KUKA KRL program: EPS_2_26115_SA7000_A_20260219035533.src

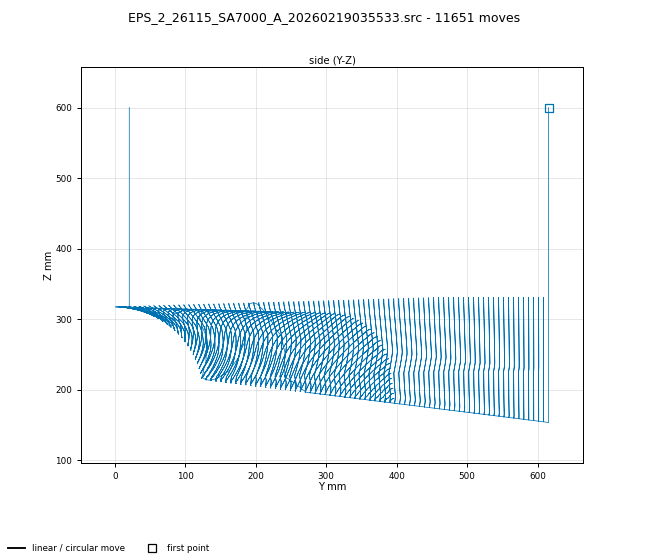
[picture p0: tool path of EPS_2_26115_SA7000_A_20260219035533.src, 11651 of 11653 moves have a stored position in this frame; points joined in program order, loops and branches not executed]
&ACCESS RVP
&REL 4
&COMMENT QRS 19112012
&PARAM EDITMASK = *
DEF PART()
EXT BAS (BAS_COMMAND :IN,REAL :IN )
INT I
BAS (#INITMOV,0 )

;KUKA QRS Post kuka4.cps  Date:22-06-2017 !

File_ID=3055

QRS_PRE_INIT()

;Init var - Until changes are made in qrs_pre_init
Outlet_Square_prg=0
Inlet_1_Square_prg=0
Inlet_2_Square_prg=0
Inlet_3_Square_prg=0
Inlet_4_Square_prg=0
Inlet_5_Square_prg=0

Outlet_1={X 0.000, Y 460.000, Z 230.500, B 0.000, E1 0.000 }
Inlet_1={X 0.000, Y 565.490, Z 205.500, B 0.000, E1 180.000 }
Outlet_1_type=201
Inlet_1_type=0
;QRS#1=Sidecore dimensions
;QRS#2=200-8" PVC SDR 35 Cut Back
;QRS#3=DeadEnd 201
;QRS#4=
;QRS#5=
;QRS#6=
;QRS#7=
;QRS#8=
;QRS#9=12-08 PSX
;QRS#10=

;QRS#11=
;QRS#12=
;QRS#13=
;QRS#14=
;QRS#15=
;QRS#16=1220x127x610 2'
;QRS#17=EPS Height
;QRS#18=331
;QRS#19=*
;QRS#20= UPDATED VERSION 22-06-2017
;QRS#21=*
Outlet_Square=0100
Inlet_1_Square=00
Inlet_2_Square=0
Inlet_3_Square=0
Inlet_4_Square=0
Inlet_5_Square=0
Mill_Square=1
Outlet_Square_Prg=214
Inlet_1_Square_prg=0

QRS_INIT()

$ADVANCE=5

; T1
PTP {E1 173.609,E2 173.609}
PTP {X 0,Y 615.488,A -85,B 0,C 180,E1 173.609,E2 173.609,E3 0,E4 0,E5 0,E6 0}
QRS_SPEED_INIT()
LIN {X 0,Y 615.488,Z 600,A -85,B 0,C 180,E1 173.609,E2 173.609,E3 0,E4 0,E5 0,E6 0} C_VEL
LIN {X 0,Y 615.488,Z 163.366,A -85,B 0,C 180,E1 173.609,E2 173.609} C_VEL
LIN {X 0,Y 615.488,Z 155.185,A -85,B 0,C 180,E1 173.609,E2 173.609} C_VEL
LIN {X 0,Y 615.477,Z 153.185,A -85,B 0,C 180,E1 173.423,E2 173.423} C_VEL
LIN {X 0,Y 615.491,Z 153.195,A -85,B 0,C 180,E1 170.802,E2 170.802} C_VEL
LIN {X 0,Y 615.463,Z 153.193,A -85,B 0,C 180,E1 168.139,E2 168.139} C_VEL
LIN {X 0,Y 615.491,Z 153.184,A -85,B 0,C 180,E1 165.451,E2 165.451} C_VEL
LIN {X 0,Y 615.488,Z 153.199,A -85,B 0,C 180,E1 162.73,E2 162.73} C_VEL
LIN {X 0,Y 615.475,Z 153.186,A -85,B 0,C 180,E1 159.967,E2 159.967} C_VEL
LIN {X 0,Y 615.485,Z 153.198,A -85,B 0,C 180,E1 157.156,E2 157.156} C_VEL
LIN {X 0,Y 615.467,Z 153.19,A -85,B 0,C 180,E1 154.433,E2 154.433} C_VEL
LIN {X 0,Y 615.482,Z 153.184,A -85,B 0,C 180,E1 152.085,E2 152.085} C_VEL
LIN {X 0,Y 615.486,Z 153.198,A -85,B 0,C 180,E1 149.081,E2 149.081} C_VEL
LIN {X 0,Y 615.474,Z 153.186,A -85,B 0,C 180,E1 146.466,E2 146.466} C_VEL
LIN {X 0,Y 615.488,Z 153.184,A -85,B 0,C 180,E1 144.165,E2 144.165} C_VEL
LIN {X 0,Y 615.484,Z 153.189,A -85,B 0,C 180,E1 141.932,E2 141.932} C_VEL
LIN {X 0,Y 615.488,Z 153.198,A -85,B 0,C 180,E1 139.394,E2 139.394} C_VEL
LIN {X 0,Y 615.477,Z 153.186,A -85,B 0,C 180,E1 136.755,E2 136.755} C_VEL
LIN {X 0,Y 615.481,Z 153.194,A -85,B 0,C 180,E1 133.997,E2 133.997} C_VEL
LIN {X 0,Y 615.478,Z 153.195,A -85,B 0,C 180,E1 131.474,E2 131.474} C_VEL
LIN {X 0,Y 615.478,Z 153.185,A -85,B 0,C 180,E1 128.904,E2 128.904} C_VEL
LIN {X 0,Y 615.483,Z 153.189,A -85,B 0,C 180,E1 126.424,E2 126.424} C_VEL
LIN {X 0,Y 615.491,Z 153.201,A -85,B 0,C 180,E1 124.021,E2 124.021} C_VEL
LIN {X 0,Y 615.481,Z 153.184,A -85,B 0,C 180,E1 121.086,E2 121.086} C_VEL
LIN {X 0,Y 615.484,Z 153.194,A -85,B 0,C 180,E1 118.451,E2 118.451} C_VEL
LIN {X 0,Y 615.472,Z 153.191,A -85,B 0,C 180,E1 115.716,E2 115.716} C_VEL
LIN {X 0,Y 615.478,Z 153.186,A -85,B 0,C 180,E1 113.556,E2 113.556} C_VEL
LIN {X 0,Y 615.482,Z 153.193,A -85,B 0,C 180,E1 110.731,E2 110.731} C_VEL
LIN {X 0,Y 615.475,Z 153.191,A -85,B 0,C 180,E1 107.957,E2 107.957} C_VEL
LIN {X 0,Y 615.484,Z 153.186,A -85,B 0,C 180,E1 105.226,E2 105.226} C_VEL
LIN {X 0,Y 615.491,Z 153.199,A -85,B 0,C 180,E1 102.53,E2 102.53} C_VEL
LIN {X 0,Y 615.486,Z 153.184,A -85,B 0,C 180,E1 99.862,E2 99.862} C_VEL
LIN {X 0,Y 615.479,Z 153.191,A -85,B 0,C 180,E1 97.216,E2 97.216} C_VEL
LIN {X 0,Y 615.482,Z 153.195,A -85,B 0,C 180,E1 94.585,E2 94.585} C_VEL
LIN {X 0,Y 615.498,Z 153.181,A -85,B 0,C 180,E1 91.963,E2 91.963} C_VEL
LIN {X 0,Y 615.481,Z 153.194,A -85,B 0,C 180,E1 89.346,E2 89.346} C_VEL
LIN {X 0,Y 615.48,Z 153.193,A -85,B 0,C 180,E1 86.727,E2 86.727} C_VEL
LIN {X 0,Y 615.492,Z 153.182,A -85,B 0,C 180,E1 84.102,E2 84.102} C_VEL
LIN {X 0,Y 615.485,Z 153.196,A -85,B 0,C 180,E1 81.463,E2 81.463} C_VEL
LIN {X 0,Y 615.48,Z 153.189,A -85,B 0,C 180,E1 78.807,E2 78.807} C_VEL
LIN {X 0,Y 615.476,Z 153.188,A -85,B 0,C 180,E1 76.07,E2 76.07} C_VEL
LIN {X 0,Y 615.487,Z 153.2,A -85,B 0,C 180,E1 73.414,E2 73.414} C_VEL
LIN {X 0,Y 615.486,Z 153.183,A -85,B 0,C 180,E1 70.662,E2 70.662} C_VEL
LIN {X 0,Y 615.483,Z 153.197,A -85,B 0,C 180,E1 67.864,E2 67.864} C_VEL
LIN {X 0,Y 615.489,Z 153.184,A -85,B 0,C 180,E1 65.009,E2 65.009} C_VEL
LIN {X 0,Y 615.488,Z 153.183,A -85,B 0,C 180,E1 62.823,E2 62.823} C_VEL
LIN {X 0,Y 615.478,Z 153.194,A -85,B 0,C 180,E1 60.206,E2 60.206} C_VEL
LIN {X 0,Y 615.482,Z 153.191,A -85,B 0,C 180,E1 57.543,E2 57.543} C_VEL
LIN {X 0,Y 615.496,Z 153.181,A -85,B 0,C 180,E1 55.186,E2 55.186} C_VEL
LIN {X 0,Y 615.473,Z 153.189,A -85,B 0,C 180,E1 52.757,E2 52.757} C_VEL
LIN {X 0,Y 615.486,Z 153.194,A -85,B 0,C 180,E1 49.911,E2 49.911} C_VEL
LIN {X 0,Y 615.487,Z 153.186,A -85,B 0,C 180,E1 47.648,E2 47.648} C_VEL
LIN {X 0,Y 615.471,Z 153.19,A -85,B 0,C 180,E1 44.931,E2 44.931} C_VEL
LIN {X 0,Y 615.485,Z 153.192,A -85,B 0,C 180,E1 42.081,E2 42.081} C_VEL
LIN {X 0,Y 615.495,Z 153.182,A -85,B 0,C 180,E1 39.749,E2 39.749} C_VEL
LIN {X 0,Y 615.474,Z 153.194,A -85,B 0,C 180,E1 36.936,E2 36.936} C_VEL
LIN {X 0,Y 615.49,Z 153.2,A -85,B 0,C 180,E1 34.702,E2 34.702} C_VEL
LIN {X 0,Y 615.479,Z 153.185,A -85,B 0,C 180,E1 31.685,E2 31.685} C_VEL
LIN {X 0,Y 615.468,Z 153.191,A -85,B 0,C 180,E1 29.407,E2 29.407} C_VEL
LIN {X 0,Y 615.484,Z 153.198,A -85,B 0,C 180,E1 27.046,E2 27.046} C_VEL
LIN {X 0,Y 615.483,Z 153.184,A -85,B 0,C 180,E1 24.009,E2 24.009} C_VEL
LIN {X 0,Y 615.471,Z 153.194,A -85,B 0,C 180,E1 21.432,E2 21.432} C_VEL
LIN {X 0,Y 615.49,Z 153.187,A -85,B 0,C 180,E1 18.608,E2 18.608} C_VEL
LIN {X 0,Y 615.466,Z 153.19,A -85,B 0,C 180,E1 15.905,E2 15.905} C_VEL
LIN {X 0,Y 615.495,Z 153.198,A -85,B 0,C 180,E1 13.201,E2 13.201} C_VEL
LIN {X 0,Y 615.483,Z 153.184,A -85,B 0,C 180,E1 10.527,E2 10.527} C_VEL
LIN {X 0,Y 615.466,Z 153.194,A -85,B 0,C 180,E1 7.876,E2 7.876} C_VEL
LIN {X 0,Y 615.49,Z 153.193,A -85,B 0,C 180,E1 5.241,E2 5.241} C_VEL
LIN {X 0,Y 615.474,Z 153.186,A -85,B 0,C 180,E1 2.618,E2 2.618} C_VEL
LIN {X 0,Y 615.473,Z 153.196,A -85,B 0,C 180,E1 0,E2 0} C_VEL
LIN {X 0,Y 615.49,Z 153.19,A -85,B 0,C 180,E1 -2.618,E2 -2.618} C_VEL
LIN {X 0,Y 615.467,Z 153.188,A -85,B 0,C 180,E1 -5.242,E2 -5.242} C_VEL
LIN {X 0,Y 615.48,Z 153.197,A -85,B 0,C 180,E1 -7.876,E2 -7.876} C_VEL
LIN {X 0,Y 615.475,Z 153.186,A -85,B 0,C 180,E1 -10.887,E2 -10.887} C_VEL
LIN {X 0,Y 615.46,Z 153.191,A -85,B 0,C 180,E1 -13.202,E2 -13.202} C_VEL
LIN {X 0,Y 615.488,Z 153.2,A -85,B 0,C 180,E1 -15.905,E2 -15.905} C_VEL
LIN {X 0,Y 615.474,Z 153.186,A -85,B 0,C 180,E1 -18.647,E2 -18.647} C_VEL
LIN {X 0,Y 615.476,Z 153.197,A -85,B 0,C 180,E1 -21.433,E2 -21.433} C_VEL
LIN {X 0,Y 615.485,Z 153.186,A -85,B 0,C 180,E1 -24.272,E2 -24.272} C_VEL
LIN {X 0,Y 615.469,Z 153.187,A -85,B 0,C 180,E1 -26.445,E2 -26.445} C_VEL
LIN {X 0,Y 615.455,Z 153.191,A -85,B 0,C 180,E1 -28.66,E2 -28.66} C_VEL
LIN {X 0,Y 615.471,Z 153.197,A -85,B 0,C 180,E1 -31.085,E2 -31.085} C_VEL
LIN {X 0,Y 615.48,Z 153.186,A -85,B 0,C 180,E1 -34.023,E2 -34.023} C_VEL
LIN {X 0,Y 615.455,Z 153.191,A -85,B 0,C 180,E1 -36.427,E2 -36.427} C_VEL
LIN {X 0,Y 615.49,Z 153.199,A -85,B 0,C 180,E1 -39.063,E2 -39.063} C_VEL
LIN {X 0,Y 615.493,Z 153.189,A -85,B 0,C 180,E1 -41.474,E2 -41.474} C_VEL
LIN {X 0,Y 615.454,Z 153.191,A -85,B 0,C 180,E1 -44.153,E2 -44.153} C_VEL
LIN {X 0,Y 615.489,Z 153.201,A -85,B 0,C 180,E1 -46.953,E2 -46.953} C_VEL
LIN {X 0,Y 615.481,Z 153.336,A -85,B 0,C 180,E1 -48.716,E2 -48.716} C_VEL
LIN {X 0,Y 615.489,Z 158.318,A -85,B 0,C 180,E1 -51.096,E2 -51.096} C_VEL
LIN {X 0,Y 615.47,Z 163.694,A -85,B 0,C 180,E1 -53.575,E2 -53.575} C_VEL
LIN {X 0,Y 615.471,Z 169.069,A -85,B 0,C 180,E1 -55.978,E2 -55.978} C_VEL
LIN {X 0,Y 615.484,Z 175.834,A -85,B 0,C 180,E1 -58.915,E2 -58.915} C_VEL
LIN {X 0,Y 615.48,Z 182.098,A -85,B 0,C 180,E1 -61.552,E2 -61.552} C_VEL
LIN {X 0,Y 615.472,Z 188.743,A -85,B 0,C 180,E1 -64.284,E2 -64.284} C_VEL
LIN {X 0,Y 615.474,Z 194.107,A -85,B 0,C 180,E1 -66.444,E2 -66.444} C_VEL
LIN {X 0,Y 615.49,Z 201.253,A -85,B 0,C 180,E1 -69.27,E2 -69.27} C_VEL
LIN {X 0,Y 615.457,Z 208.403,A -85,B 0,C 180,E1 -72.042,E2 -72.042} C_VEL
LIN {X 0,Y 615.495,Z 215.538,A -85,B 0,C 180,E1 -74.774,E2 -74.774} C_VEL
LIN {X 0,Y 615.438,Z 222.684,A -85,B 0,C 180,E1 -77.469,E2 -77.469} C_VEL
LIN {X 0,Y 615.49,Z 225.076,A -85,B 0,C 180,E1 -78.369,E2 -78.369} C_VEL
LIN {X 0,Y 615.481,Z 240.867,A -85,B 0,C 180,E1 -78.724,E2 -78.724} C_VEL
LIN {X 0,Y 615.44,Z 253.271,A -85,B 0,C 180,E1 -79.136,E2 -79.136} C_VEL
LIN {X 0,Y 615.434,Z 264.489,A -85,B 0,C 180,E1 -79.639,E2 -79.639} C_VEL
LIN {X 0,Y 615.485,Z 275.998,A -85,B 0,C 180,E1 -80.304,E2 -80.304} C_VEL
LIN {X 0,Y 615.499,Z 286.343,A -85,B 0,C 180,E1 -81.05,E2 -81.05} C_VEL
LIN {X 0,Y 615.497,Z 294.813,A -85,B 0,C 180,E1 -81.794,E2 -81.794} C_VEL
LIN {X 0,Y 615.498,Z 302.607,A -85,B 0,C 180,E1 -82.62,E2 -82.62} C_VEL
LIN {X 0,Y 615.496,Z 310.204,A -85,B 0,C 180,E1 -83.608,E2 -83.608} C_VEL
LIN {X 0,Y 615.498,Z 317.205,A -85,B 0,C 180,E1 -84.759,E2 -84.759} C_VEL
LIN {X 0,Y 615.493,Z 321.852,A -85,B 0,C 180,E1 -85.744,E2 -85.744} C_VEL
LIN {X 0,Y 615.494,Z 325.399,A -85,B 0,C 180,E1 -86.727,E2 -86.727} C_VEL
LIN {X 0,Y 615.497,Z 327.233,A -85,B 0,C 180,E1 -87.382,E2 -87.382} C_VEL
LIN {X 0,Y 615.5,Z 328.608,A -85,B 0,C 180,E1 -88.037,E2 -88.037} C_VEL
LIN {X 0,Y 615.496,Z 330.173,A -85,B 0,C 180,E1 -89.346,E2 -89.346} C_VEL
LIN {X 0,Y 615.494,Z 330.389,A -85,B 0,C 180,E1 -90,E2 -90} C_VEL
LIN {X 0,Y 615.495,Z 329.58,A -85,B 0,C 180,E1 -91.309,E2 -91.309} C_VEL
LIN {X 0,Y 615.5,Z 328.608,A -85,B 0,C 180,E1 -91.963,E2 -91.963} C_VEL
LIN {X 0,Y 615.497,Z 327.233,A -85,B 0,C 180,E1 -92.618,E2 -92.618} C_VEL
LIN {X 0,Y 615.496,Z 324.35,A -85,B 0,C 180,E1 -93.601,E2 -93.601} C_VEL
LIN {X 0,Y 615.498,Z 320.442,A -85,B 0,C 180,E1 -94.584,E2 -94.584} C_VEL
LIN {X 0,Y 615.499,Z 315.405,A -85,B 0,C 180,E1 -95.57,E2 -95.57} C_VEL
LIN {X 0,Y 615.497,Z 308.87,A -85,B 0,C 180,E1 -96.583,E2 -96.583} C_VEL
LIN {X 0,Y 615.497,Z 301.134,A -85,B 0,C 180,E1 -97.545,E2 -97.545} C_VEL
LIN {X 0,Y 615.498,Z 293.046,A -85,B 0,C 180,E1 -98.371,E2 -98.371} C_VEL
LIN {X 0,Y 615.499,Z 283.169,A -85,B 0,C 180,E1 -99.198,E2 -99.198} C_VEL
LIN {X 0,Y 615.464,Z 271.988,A -85,B 0,C 180,E1 -99.945,E2 -99.945} C_VEL
LIN {X 0,Y 615.43,Z 261.035,A -85,B 0,C 180,E1 -100.528,E2 -100.528} C_VEL
LIN {X 0,Y 615.453,Z 248.835,A -85,B 0,C 180,E1 -101.029,E2 -101.029} C_VEL
LIN {X 0,Y 615.495,Z 236.071,A -85,B 0,C 180,E1 -101.401,E2 -101.401} C_VEL
LIN {X 0,Y 615.49,Z 225.076,A -85,B 0,C 180,E1 -101.631,E2 -101.631} C_VEL
LIN {X 0,Y 615.457,Z 219,A -85,B 0,C 180,E1 -103.92,E2 -103.92} C_VEL
LIN {X 0,Y 615.451,Z 212.413,A -85,B 0,C 180,E1 -106.419,E2 -106.419} C_VEL
LIN {X 0,Y 615.487,Z 204.835,A -85,B 0,C 180,E1 -109.338,E2 -109.338} C_VEL
LIN {X 0,Y 615.47,Z 197.68,A -85,B 0,C 180,E1 -112.137,E2 -112.137} C_VEL
LIN {X 0,Y 615.49,Z 190.536,A -85,B 0,C 180,E1 -114.991,E2 -114.991} C_VEL
LIN {X 0,Y 615.489,Z 185.167,A -85,B 0,C 180,E1 -117.177,E2 -117.177} C_VEL
LIN {X 0,Y 615.49,Z 178.875,A -85,B 0,C 180,E1 -119.794,E2 -119.794} C_VEL
LIN {X 0,Y 615.471,Z 172.648,A -85,B 0,C 180,E1 -122.458,E2 -122.458} C_VEL
LIN {X 0,Y 615.496,Z 167.272,A -85,B 0,C 180,E1 -124.814,E2 -124.814} C_VEL
LIN {X 0,Y 615.489,Z 161.901,A -85,B 0,C 180,E1 -127.241,E2 -127.241} C_VEL
LIN {X 0,Y 615.454,Z 156.533,A -85,B 0,C 180,E1 -129.752,E2 -129.752} C_VEL
LIN {X 0,Y 615.474,Z 153.198,A -85,B 0,C 180,E1 -131.379,E2 -131.379} C_VEL
LIN {X 0,Y 615.461,Z 153.189,A -85,B 0,C 180,E1 -134.151,E2 -134.151} C_VEL
LIN {X 0,Y 615.487,Z 153.202,A -85,B 0,C 180,E1 -136.952,E2 -136.952} C_VEL
LIN {X 0,Y 615.459,Z 153.195,A -85,B 0,C 180,E1 -139.391,E2 -139.391} C_VEL
LIN {X 0,Y 615.472,Z 153.187,A -85,B 0,C 180,E1 -141.989,E2 -141.989} C_VEL
LIN {X 0,Y 615.493,Z 153.19,A -85,B 0,C 180,E1 -144.384,E2 -144.384} C_VEL
LIN {X 0,Y 615.485,Z 153.2,A -85,B 0,C 180,E1 -146.763,E2 -146.763} C_VEL
LIN {X 0,Y 615.461,Z 153.195,A -85,B 0,C 180,E1 -149.078,E2 -149.078} C_VEL
LIN {X 0,Y 615.464,Z 153.188,A -85,B 0,C 180,E1 -151.552,E2 -151.552} C_VEL
LIN {X 0,Y 615.499,Z 153.2,A -85,B 0,C 180,E1 -154.427,E2 -154.427} C_VEL
LIN {X 0,Y 615.458,Z 153.191,A -85,B 0,C 180,E1 -157.154,E2 -157.154} C_VEL
LIN {X 0,Y 615.492,Z 153.191,A -85,B 0,C 180,E1 -159.967,E2 -159.967} C_VEL
LIN {X 0,Y 615.461,Z 153.193,A -85,B 0,C 180,E1 -162.728,E2 -162.728} C_VEL
LIN {X 0,Y 615.489,Z 153.185,A -85,B 0,C 180,E1 -165.451,E2 -165.451} C_VEL
LIN {X 0,Y 615.483,Z 153.2,A -85,B 0,C 180,E1 -168.139,E2 -168.139} C_VEL
LIN {X 0,Y 615.463,Z 153.189,A -85,B 0,C 180,E1 -170.801,E2 -170.801} C_VEL
LIN {X 0,Y 615.489,Z 153.189,A -85,B 0,C 180,E1 -173.443,E2 -173.443} C_VEL
LIN {X 0,Y 615.475,Z 153.196,A -85,B 0,C 180,E1 -176.071,E2 -176.071} C_VEL
LIN {X 0,Y 615.47,Z 153.187,A -85,B 0,C 180,E1 -178.691,E2 -178.691} C_VEL
LIN {X 0,Y 615.488,Z 153.192,A -85,B 0,C 180,E1 -181.308,E2 -181.308} C_VEL
LIN {X 0,Y 615.471,Z 153.195,A -85,B 0,C 180,E1 -183.928,E2 -183.928} C_VEL
LIN {X 0,Y 615.477,Z 153.185,A -85,B 0,C 180,E1 -186.577,E2 -186.577} C_VEL
LIN {X 0,Y 614.811,Z 153.341,A -85,B 0,C 180,E1 -187.123,E2 -187.123} C_VEL
LIN {X 0,Y 611.986,Z 153.75,A -85,B 0,C 180,E1 -188.009,E2 -188.009} C_VEL
LIN {X 0,Y 609.592,Z 154.065,A -85,B 0,C 180,E1 -188.722,E2 -188.722} C_VEL
LIN {X 0,Y 608.549,Z 154.185,A -85,B 0,C 180,E1 -189.272,E2 -189.272} C_VEL
LIN {X 0,Y 608.456,Z 154.193,A -85,B 0,C 180,E1 -189.458,E2 -189.458} C_VEL
LIN {X 0,Y 608.446,Z 154.19,A -85,B 0,C 180,E1 -192,E2 -192} C_VEL
LIN {X 0,Y 608.478,Z 154.187,A -85,B 0,C 180,E1 -194.72,E2 -194.72} C_VEL
LIN {X 0,Y 608.448,Z 154.193,A -85,B 0,C 180,E1 -197.476,E2 -197.476} C_VEL
LIN {X 0,Y 608.458,Z 154.187,A -85,B 0,C 180,E1 -200.274,E2 -200.274} C_VEL
LIN {X 0,Y 608.442,Z 154.197,A -85,B 0,C 180,E1 -203.124,E2 -203.124} C_VEL
LIN {X 0,Y 608.456,Z 154.188,A -85,B 0,C 180,E1 -205.72,E2 -205.72} C_VEL
LIN {X 0,Y 608.449,Z 154.19,A -85,B 0,C 180,E1 -208.266,E2 -208.266} C_VEL
LIN {X 0,Y 608.472,Z 154.192,A -85,B 0,C 180,E1 -210.544,E2 -210.544} C_VEL
LIN {X 0,Y 608.449,Z 154.195,A -85,B 0,C 180,E1 -212.88,E2 -212.88} C_VEL
LIN {X 0,Y 608.439,Z 154.191,A -85,B 0,C 180,E1 -215.277,E2 -215.277} C_VEL
LIN {X 0,Y 608.463,Z 154.192,A -85,B 0,C 180,E1 -218.241,E2 -218.241} C_VEL
LIN {X 0,Y 608.475,Z 154.193,A -85,B 0,C 180,E1 -220.333,E2 -220.333} C_VEL
LIN {X 0,Y 608.465,Z 154.186,A -85,B 0,C 180,E1 -223.309,E2 -223.309} C_VEL
LIN {X 0,Y 608.465,Z 154.193,A -85,B 0,C 180,E1 -226.131,E2 -226.131} C_VEL
LIN {X 0,Y 608.443,Z 154.191,A -85,B 0,C 180,E1 -228.823,E2 -228.823} C_VEL
LIN {X 0,Y 608.463,Z 154.187,A -85,B 0,C 180,E1 -231.412,E2 -231.412} C_VEL
LIN {X 0,Y 608.475,Z 154.193,A -85,B 0,C 180,E1 -233.95,E2 -233.95} C_VEL
LIN {X 0,Y 608.457,Z 154.192,A -85,B 0,C 180,E1 -236.329,E2 -236.329} C_VEL
LIN {X 0,Y 608.472,Z 154.186,A -85,B 0,C 180,E1 -238.728,E2 -238.728} C_VEL
LIN {X 0,Y 608.47,Z 154.188,A -85,B 0,C 180,E1 -241.38,E2 -241.38} C_VEL
LIN {X 0,Y 608.438,Z 154.197,A -85,B 0,C 180,E1 -243.965,E2 -243.965} C_VEL
LIN {X 0,Y 608.461,Z 154.19,A -85,B 0,C 180,E1 -246.155,E2 -246.155} C_VEL
LIN {X 0,Y 608.468,Z 154.187,A -85,B 0,C 180,E1 -248.309,E2 -248.309} C_VEL
LIN {X 0,Y 608.471,Z 154.191,A -85,B 0,C 180,E1 -251.283,E2 -251.283} C_VEL
LIN {X 0,Y 608.455,Z 154.191,A -85,B 0,C 180,E1 -253.906,E2 -253.906} C_VEL
LIN {X 0,Y 608.458,Z 154.188,A -85,B 0,C 180,E1 -256.644,E2 -256.644} C_VEL
LIN {X 0,Y 608.464,Z 154.197,A -85,B 0,C 180,E1 -259.35,E2 -259.35} C_VEL
LIN {X 0,Y 608.476,Z 154.185,A -85,B 0,C 180,E1 -262.033,E2 -262.033} C_VEL
LIN {X 0,Y 608.46,Z 154.19,A -85,B 0,C 180,E1 -264.698,E2 -264.698} C_VEL
LIN {X 0,Y 608.472,Z 154.191,A -85,B 0,C 180,E1 -267.352,E2 -267.352} C_VEL
LIN {X 0,Y 608.477,Z 154.185,A -85,B 0,C 180,E1 -270,E2 -270} C_VEL
LIN {X 0,Y 608.472,Z 154.191,A -85,B 0,C 180,E1 -272.648,E2 -272.648} C_VEL
LIN {X 0,Y 608.46,Z 154.19,A -85,B 0,C 180,E1 -275.302,E2 -275.302} C_VEL
LIN {X 0,Y 608.476,Z 154.185,A -85,B 0,C 180,E1 -277.967,E2 -277.967} C_VEL
LIN {X 0,Y 608.467,Z 154.191,A -85,B 0,C 180,E1 -280.957,E2 -280.957} C_VEL
LIN {X 0,Y 608.458,Z 154.188,A -85,B 0,C 180,E1 -283.356,E2 -283.356} C_VEL
LIN {X 0,Y 608.455,Z 154.191,A -85,B 0,C 180,E1 -286.094,E2 -286.094} C_VEL
LIN {X 0,Y 608.455,Z 154.191,A -85,B 0,C 180,E1 -288.869,E2 -288.869} C_VEL
LIN {X 0,Y 608.468,Z 154.187,A -85,B 0,C 180,E1 -291.691,E2 -291.691} C_VEL
LIN {X 0,Y 608.454,Z 154.193,A -85,B 0,C 180,E1 -294.571,E2 -294.571} C_VEL
LIN {X 0,Y 608.448,Z 154.189,A -85,B 0,C 180,E1 -297.518,E2 -297.518} C_VEL
LIN {X 0,Y 608.464,Z 154.194,A -85,B 0,C 180,E1 -299.972,E2 -299.972} C_VEL
LIN {X 0,Y 608.457,Z 154.19,A -85,B 0,C 180,E1 -302.522,E2 -302.522} C_VEL
LIN {X 0,Y 608.441,Z 154.19,A -85,B 0,C 180,E1 -305.277,E2 -305.277} C_VEL
LIN {X 0,Y 608.465,Z 154.19,A -85,B 0,C 180,E1 -308.241,E2 -308.241} C_VEL
LIN {X 0,Y 608.476,Z 154.187,A -85,B 0,C 180,E1 -310.332,E2 -310.332} C_VEL
LIN {X 0,Y 608.461,Z 154.19,A -85,B 0,C 180,E1 -313.309,E2 -313.309} C_VEL
LIN {X 0,Y 608.468,Z 154.188,A -85,B 0,C 180,E1 -316.131,E2 -316.131} C_VEL
LIN {X 0,Y 608.443,Z 154.19,A -85,B 0,C 180,E1 -318.823,E2 -318.823} C_VEL
LIN {X 0,Y 608.461,Z 154.196,A -85,B 0,C 180,E1 -321.412,E2 -321.412} C_VEL
LIN {X 0,Y 608.474,Z 154.187,A -85,B 0,C 180,E1 -323.95,E2 -323.95} C_VEL
LIN {X 0,Y 608.456,Z 154.187,A -85,B 0,C 180,E1 -326.329,E2 -326.329} C_VEL
LIN {X 0,Y 608.452,Z 154.19,A -85,B 0,C 180,E1 -328.73,E2 -328.73} C_VEL
LIN {X 0,Y 608.472,Z 154.192,A -85,B 0,C 180,E1 -331.379,E2 -331.379} C_VEL
LIN {X 0,Y 608.436,Z 154.19,A -85,B 0,C 180,E1 -333.965,E2 -333.965} C_VEL
LIN {X 0,Y 608.458,Z 154.187,A -85,B 0,C 180,E1 -336.155,E2 -336.155} C_VEL
LIN {X 0,Y 608.459,Z 154.188,A -85,B 0,C 180,E1 -338.309,E2 -338.309} C_VEL
LIN {X 0,Y 608.47,Z 154.189,A -85,B 0,C 180,E1 -341.282,E2 -341.282} C_VEL
LIN {X 0,Y 608.449,Z 154.188,A -85,B 0,C 180,E1 -343.906,E2 -343.906} C_VEL
LIN {X 0,Y 608.465,Z 154.196,A -85,B 0,C 180,E1 -346.644,E2 -346.644} C_VEL
LIN {X 0,Y 608.463,Z 154.187,A -85,B 0,C 180,E1 -349.351,E2 -349.351} C_VEL
LIN {X 0,Y 608.462,Z 154.189,A -85,B 0,C 180,E1 -352.033,E2 -352.033} C_VEL
LIN {X 0,Y 608.466,Z 154.192,A -85,B 0,C 180,E1 -354.699,E2 -354.699} C_VEL
LIN {X 0,Y 608.466,Z 154.186,A -85,B 0,C 180,E1 -357.352,E2 -357.352} C_VEL
LIN {X 0,Y 608.464,Z 154.191,A -85,B 0,C 180,E1 -360,E2 -360} C_VEL
LIN {X 0,Y 608.479,Z 154.188,A -85,B 0,C 180,E1 -362.648,E2 -362.648} C_VEL
LIN {X 0,Y 608.448,Z 154.188,A -85,B 0,C 180,E1 -365.302,E2 -365.302} C_VEL
LIN {X 0,Y 608.473,Z 154.194,A -85,B 0,C 180,E1 -367.967,E2 -367.967} C_VEL
LIN {X 0,Y 608.461,Z 154.186,A -85,B 0,C 180,E1 -370.956,E2 -370.956} C_VEL
LIN {X 0,Y 608.446,Z 154.19,A -85,B 0,C 180,E1 -373.357,E2 -373.357} C_VEL
LIN {X 0,Y 608.463,Z 154.192,A -85,B 0,C 180,E1 -376.094,E2 -376.094} C_VEL
LIN {X 0,Y 608.445,Z 154.189,A -85,B 0,C 180,E1 -378.87,E2 -378.87} C_VEL
LIN {X 0,Y 608.464,Z 154.196,A -85,B 0,C 180,E1 -381.692,E2 -381.692} C_VEL
LIN {X 0,Y 608.442,Z 154.189,A -85,B 0,C 180,E1 -384.572,E2 -384.572} C_VEL
LIN {X 0,Y 608.464,Z 154.192,A -85,B 0,C 180,E1 -387.206,E2 -387.206} C_VEL
LIN {X 0,Y 608.47,Z 154.188,A -85,B 0,C 180,E1 -389.973,E2 -389.973} C_VEL
LIN {X 0,Y 608.445,Z 154.192,A -85,B 0,C 180,E1 -392.881,E2 -392.881} C_VEL
LIN {X 0,Y 608.436,Z 154.2,A -85,B 0,C 180,E1 -395.278,E2 -395.278} C_VEL
LIN {X 0,Y 608.462,Z 154.189,A -85,B 0,C 180,E1 -397.747,E2 -397.747} C_VEL
LIN {X 0,Y 608.429,Z 154.191,A -85,B 0,C 180,E1 -400.327,E2 -400.327} C_VEL
LIN {X 0,Y 608.449,Z 154.198,A -85,B 0,C 180,E1 -402.961,E2 -402.961} C_VEL
LIN {X 0,Y 608.436,Z 154.191,A -85,B 0,C 180,E1 -405.738,E2 -405.738} C_VEL
LIN {X 0,Y 608.461,Z 154.31,A -85,B 0,C 180,E1 -408.524,E2 -408.524} C_VEL
LIN {X 0,Y 608.472,Z 158.676,A -85,B 0,C 180,E1 -410.703,E2 -410.703} C_VEL
LIN {X 0,Y 608.472,Z 163.769,A -85,B 0,C 180,E1 -413.087,E2 -413.087} C_VEL
LIN {X 0,Y 608.466,Z 169.158,A -85,B 0,C 180,E1 -415.531,E2 -415.531} C_VEL
LIN {X 0,Y 608.458,Z 174.548,A -85,B 0,C 180,E1 -417.906,E2 -417.906} C_VEL
LIN {X 0,Y 608.474,Z 179.937,A -85,B 0,C 180,E1 -420.221,E2 -420.221} C_VEL
LIN {X 0,Y 608.462,Z 186.082,A -85,B 0,C 180,E1 -422.796,E2 -422.796} C_VEL
LIN {X 0,Y 608.456,Z 192.513,A -85,B 0,C 180,E1 -425.429,E2 -425.429} C_VEL
LIN {X 0,Y 608.437,Z 199.699,A -85,B 0,C 180,E1 -428.308,E2 -428.308} C_VEL
LIN {X 0,Y 608.445,Z 205.089,A -85,B 0,C 180,E1 -430.43,E2 -430.43} C_VEL
LIN {X 0,Y 608.419,Z 212.275,A -85,B 0,C 180,E1 -433.215,E2 -433.215} C_VEL
LIN {X 0,Y 608.393,Z 217.664,A -85,B 0,C 180,E1 -435.278,E2 -435.278} C_VEL
LIN {X 0,Y 608.381,Z 223.054,A -85,B 0,C 180,E1 -437.321,E2 -437.321} C_VEL
LIN {X 0,Y 608.451,Z 225.628,A -85,B 0,C 180,E1 -438.254,E2 -438.254} C_VEL
LIN {X 0,Y 608.542,Z 238.707,A -85,B 0,C 180,E1 -438.53,E2 -438.53} C_VEL
LIN {X 0,Y 608.471,Z 251.582,A -85,B 0,C 180,E1 -438.942,E2 -438.942} C_VEL
LIN {X 0,Y 608.461,Z 262.925,A -85,B 0,C 180,E1 -439.434,E2 -439.434} C_VEL
LIN {X 0,Y 608.463,Z 273.581,A -85,B 0,C 180,E1 -440.023,E2 -440.023} C_VEL
LIN {X 0,Y 608.483,Z 284.476,A -85,B 0,C 180,E1 -440.778,E2 -440.778} C_VEL
LIN {X 0,Y 608.475,Z 295.114,A -85,B 0,C 180,E1 -441.699,E2 -441.699} C_VEL
LIN {X 0,Y 608.471,Z 302.961,A -85,B 0,C 180,E1 -442.534,E2 -442.534} C_VEL
LIN {X 0,Y 608.461,Z 310.287,A -85,B 0,C 180,E1 -443.485,E2 -443.485} C_VEL
LIN {X 0,Y 608.45,Z 315.866,A -85,B 0,C 180,E1 -444.366,E2 -444.366} C_VEL
LIN {X 0,Y 608.432,Z 320.951,A -85,B 0,C 180,E1 -445.362,E2 -445.362} C_VEL
LIN {X 0,Y 608.449,Z 324.896,A -85,B 0,C 180,E1 -446.358,E2 -446.358} C_VEL
LIN {X 0,Y 608.425,Z 327.809,A -85,B 0,C 180,E1 -447.352,E2 -447.352} C_VEL
LIN {X 0,Y 608.444,Z 329.201,A -85,B 0,C 180,E1 -448.014,E2 -448.014} C_VEL
LIN {X 0,Y 608.438,Z 330.783,A -85,B 0,C 180,E1 -449.338,E2 -449.338} C_VEL
LIN {X 0,Y 608.434,Z 330.999,A -85,B 0,C 180,E1 -450,E2 -450} C_VEL
LIN {X 0,Y 608.448,Z 330.184,A -85,B 0,C 180,E1 -451.324,E2 -451.324} C_VEL
LIN {X 0,Y 608.444,Z 329.201,A -85,B 0,C 180,E1 -451.986,E2 -451.986} C_VEL
LIN {X 0,Y 608.425,Z 327.809,A -85,B 0,C 180,E1 -452.648,E2 -452.648} C_VEL
LIN {X 0,Y 608.449,Z 324.896,A -85,B 0,C 180,E1 -453.642,E2 -453.642} C_VEL
LIN {X 0,Y 608.432,Z 320.951,A -85,B 0,C 180,E1 -454.638,E2 -454.638} C_VEL
LIN {X 0,Y 608.437,Z 314.877,A -85,B 0,C 180,E1 -455.801,E2 -455.801} C_VEL
LIN {X 0,Y 608.462,Z 308.236,A -85,B 0,C 180,E1 -456.799,E2 -456.799} C_VEL
LIN {X 0,Y 608.456,Z 299.991,A -85,B 0,C 180,E1 -457.8,E2 -457.8} C_VEL
LIN {X 0,Y 608.472,Z 291.534,A -85,B 0,C 180,E1 -458.636,E2 -458.636} C_VEL
LIN {X 0,Y 608.48,Z 281.091,A -85,B 0,C 180,E1 -459.473,E2 -459.473} C_VEL
LIN {X 0,Y 608.458,Z 270.758,A -85,B 0,C 180,E1 -460.145,E2 -460.145} C_VEL
LIN {X 0,Y 608.457,Z 259.905,A -85,B 0,C 180,E1 -460.711,E2 -460.711} C_VEL
LIN {X 0,Y 608.488,Z 248.118,A -85,B 0,C 180,E1 -461.185,E2 -461.185} C_VEL
LIN {X 0,Y 608.546,Z 235.271,A -85,B 0,C 180,E1 -461.554,E2 -461.554} C_VEL
LIN {X 0,Y 608.428,Z 225.468,A -85,B 0,C 180,E1 -461.768,E2 -461.768} C_VEL
LIN {X 0,Y 608.4,Z 219.461,A -85,B 0,C 180,E1 -464.039,E2 -464.039} C_VEL
LIN {X 0,Y 608.4,Z 213,A -85,B 0,C 180,E1 -466.506,E2 -466.506} C_VEL
LIN {X 0,Y 608.429,Z 206.885,A -85,B 0,C 180,E1 -468.87,E2 -468.87} C_VEL
LIN {X 0,Y 608.458,Z 201.495,A -85,B 0,C 180,E1 -470.981,E2 -470.981} C_VEL
LIN {X 0,Y 608.454,Z 194.309,A -85,B 0,C 180,E1 -473.845,E2 -473.845} C_VEL
LIN {X 0,Y 608.448,Z 187.123,A -85,B 0,C 180,E1 -476.774,E2 -476.774} C_VEL
LIN {X 0,Y 608.437,Z 181.734,A -85,B 0,C 180,E1 -479.021,E2 -479.021} C_VEL
LIN {X 0,Y 608.477,Z 176.344,A -85,B 0,C 180,E1 -481.315,E2 -481.315} C_VEL
LIN {X 0,Y 608.472,Z 170.809,A -85,B 0,C 180,E1 -483.734,E2 -483.734} C_VEL
LIN {X 0,Y 608.471,Z 165.565,A -85,B 0,C 180,E1 -486.09,E2 -486.09} C_VEL
LIN {X 0,Y 608.462,Z 160.176,A -85,B 0,C 180,E1 -488.588,E2 -488.588} C_VEL
LIN {X 0,Y 608.522,Z 154.526,A -85,B 0,C 180,E1 -491.348,E2 -491.348} C_VEL
LIN {X 0,Y 608.438,Z 154.192,A -85,B 0,C 180,E1 -492.062,E2 -492.062} C_VEL
LIN {X 0,Y 608.459,Z 154.194,A -85,B 0,C 180,E1 -494.795,E2 -494.795} C_VEL
LIN {X 0,Y 608.449,Z 154.198,A -85,B 0,C 180,E1 -497.039,E2 -497.039} C_VEL
LIN {X 0,Y 608.449,Z 154.189,A -85,B 0,C 180,E1 -499.696,E2 -499.696} C_VEL
LIN {X 0,Y 608.462,Z 154.189,A -85,B 0,C 180,E1 -502.253,E2 -502.253} C_VEL
LIN {X 0,Y 608.43,Z 154.195,A -85,B 0,C 180,E1 -505.096,E2 -505.096} C_VEL
LIN {X 0,Y 608.434,Z 154.19,A -85,B 0,C 180,E1 -507.48,E2 -507.48} C_VEL
LIN {X 0,Y 608.477,Z 154.189,A -85,B 0,C 180,E1 -510.221,E2 -510.221} C_VEL
LIN {X 0,Y 608.428,Z 154.191,A -85,B 0,C 180,E1 -513.224,E2 -513.224} C_VEL
LIN {X 0,Y 608.482,Z 154.186,A -85,B 0,C 180,E1 -515.845,E2 -515.845} C_VEL
LIN {X 0,Y 608.464,Z 154.196,A -85,B 0,C 180,E1 -518.308,E2 -518.308} C_VEL
LIN {X 0,Y 608.445,Z 154.189,A -85,B 0,C 180,E1 -521.13,E2 -521.13} C_VEL
LIN {X 0,Y 608.463,Z 154.192,A -85,B 0,C 180,E1 -523.906,E2 -523.906} C_VEL
LIN {X 0,Y 608.446,Z 154.19,A -85,B 0,C 180,E1 -526.643,E2 -526.643} C_VEL
LIN {X 0,Y 608.463,Z 154.188,A -85,B 0,C 180,E1 -529.35,E2 -529.35} C_VEL
LIN {X 0,Y 608.473,Z 154.194,A -85,B 0,C 180,E1 -532.033,E2 -532.033} C_VEL
LIN {X 0,Y 608.448,Z 154.188,A -85,B 0,C 180,E1 -534.698,E2 -534.698} C_VEL
LIN {X 0,Y 608.479,Z 154.188,A -85,B 0,C 180,E1 -537.352,E2 -537.352} C_VEL
LIN {X 0,Y 608.464,Z 154.191,A -85,B 0,C 180,E1 -540,E2 -540} C_VEL
LIN {X 0,Y 608.466,Z 154.186,A -85,B 0,C 180,E1 -542.648,E2 -542.648} C_VEL
LIN {X 0,Y 608.466,Z 154.192,A -85,B 0,C 180,E1 -545.301,E2 -545.301} C_VEL
LIN {X 0,Y 608.462,Z 154.189,A -85,B 0,C 180,E1 -547.967,E2 -547.967} C_VEL
LIN {X 0,Y 608.456,Z 154.193,A -85,B 0,C 180,E1 -549.458,E2 -549.458} C_VEL
LIN {X 0,Y 607.766,Z 154.276,A -85,B 0,C 180,E1 -550.01,E2 -550.01} C_VEL
LIN {X 0,Y 604.904,Z 154.633,A -85,B 0,C 180,E1 -550.907,E2 -550.907} C_VEL
LIN {X 0,Y 602.506,Z 154.934,A -85,B 0,C 180,E1 -551.629,E2 -551.629} C_VEL
LIN {X 0,Y 601.483,Z 155.056,A -85,B 0,C 180,E1 -552.185,E2 -552.185} C_VEL
LIN {X 0,Y 601.403,Z 155.066,A -85,B 0,C 180,E1 -552.374,E2 -552.374} C_VEL
LIN {X 0,Y 601.43,Z 155.067,A -85,B 0,C 180,E1 -554.896,E2 -554.896} C_VEL
LIN {X 0,Y 601.429,Z 155.07,A -85,B 0,C 180,E1 -556.986,E2 -556.986} C_VEL
LIN {X 0,Y 601.4,Z 155.067,A -85,B 0,C 180,E1 -559.809,E2 -559.809} C_VEL
LIN {X 0,Y 601.409,Z 155.069,A -85,B 0,C 180,E1 -562.606,E2 -562.606} C_VEL
LIN {X 0,Y 601.399,Z 155.076,A -85,B 0,C 180,E1 -564.878,E2 -564.878} C_VEL
LIN {X 0,Y 601.416,Z 155.064,A -85,B 0,C 180,E1 -567.867,E2 -567.867} C_VEL
LIN {X 0,Y 601.442,Z 155.063,A -85,B 0,C 180,E1 -570.163,E2 -570.163} C_VEL
LIN {X 0,Y 601.418,Z 155.075,A -85,B 0,C 180,E1 -572.716,E2 -572.716} C_VEL
LIN {X 0,Y 601.407,Z 155.068,A -85,B 0,C 180,E1 -575.115,E2 -575.115} C_VEL
LIN {X 0,Y 601.427,Z 155.063,A -85,B 0,C 180,E1 -577.419,E2 -577.419} C_VEL
LIN {X 0,Y 601.408,Z 155.068,A -85,B 0,C 180,E1 -579.995,E2 -579.995} C_VEL
LIN {X 0,Y 601.407,Z 155.071,A -85,B 0,C 180,E1 -582.67,E2 -582.67} C_VEL
LIN {X 0,Y 601.419,Z 155.064,A -85,B 0,C 180,E1 -585.482,E2 -585.482} C_VEL
LIN {X 0,Y 601.417,Z 155.072,A -85,B 0,C 180,E1 -588.407,E2 -588.407} C_VEL
LIN {X 0,Y 601.429,Z 155.064,A -85,B 0,C 180,E1 -590.876,E2 -590.876} C_VEL
LIN {X 0,Y 601.44,Z 155.066,A -85,B 0,C 180,E1 -593.734,E2 -593.734} C_VEL
LIN {X 0,Y 601.427,Z 155.072,A -85,B 0,C 180,E1 -596.064,E2 -596.064} C_VEL
LIN {X 0,Y 601.436,Z 155.063,A -85,B 0,C 180,E1 -598.542,E2 -598.542} C_VEL
LIN {X 0,Y 601.43,Z 155.065,A -85,B 0,C 180,E1 -601.374,E2 -601.374} C_VEL
LIN {X 0,Y 601.401,Z 155.074,A -85,B 0,C 180,E1 -603.637,E2 -603.637} C_VEL
LIN {X 0,Y 601.415,Z 155.064,A -85,B 0,C 180,E1 -606.59,E2 -606.59} C_VEL
LIN {X 0,Y 601.43,Z 155.071,A -85,B 0,C 180,E1 -609.478,E2 -609.478} C_VEL
LIN {X 0,Y 601.395,Z 155.068,A -85,B 0,C 180,E1 -612.312,E2 -612.312} C_VEL
LIN {X 0,Y 601.41,Z 155.065,A -85,B 0,C 180,E1 -614.409,E2 -614.409} C_VEL
LIN {X 0,Y 601.421,Z 155.071,A -85,B 0,C 180,E1 -617.172,E2 -617.172} C_VEL
LIN {X 0,Y 601.433,Z 155.064,A -85,B 0,C 180,E1 -619.905,E2 -619.905} C_VEL
LIN {X 0,Y 601.437,Z 155.064,A -85,B 0,C 180,E1 -622.615,E2 -622.615} C_VEL
LIN {X 0,Y 601.419,Z 155.072,A -85,B 0,C 180,E1 -625.308,E2 -625.308} C_VEL
LIN {X 0,Y 601.436,Z 155.062,A -85,B 0,C 180,E1 -627.991,E2 -627.991} C_VEL
LIN {X 0,Y 601.447,Z 155.066,A -85,B 0,C 180,E1 -630.67,E2 -630.67} C_VEL
LIN {X 0,Y 601.426,Z 155.067,A -85,B 0,C 180,E1 -633.35,E2 -633.35} C_VEL
LIN {X 0,Y 601.437,Z 155.062,A -85,B 0,C 180,E1 -636.037,E2 -636.037} C_VEL
LIN {X 0,Y 601.434,Z 155.073,A -85,B 0,C 180,E1 -638.738,E2 -638.738} C_VEL
LIN {X 0,Y 601.431,Z 155.063,A -85,B 0,C 180,E1 -641.458,E2 -641.458} C_VEL
LIN {X 0,Y 601.416,Z 155.069,A -85,B 0,C 180,E1 -644.205,E2 -644.205} C_VEL
LIN {X 0,Y 601.431,Z 155.065,A -85,B 0,C 180,E1 -646.986,E2 -646.986} C_VEL
LIN {X 0,Y 601.403,Z 155.067,A -85,B 0,C 180,E1 -649.809,E2 -649.809} C_VEL
LIN {X 0,Y 601.411,Z 155.07,A -85,B 0,C 180,E1 -652.605,E2 -652.605} C_VEL
LIN {X 0,Y 601.4,Z 155.068,A -85,B 0,C 180,E1 -654.878,E2 -654.878} C_VEL
LIN {X 0,Y 601.418,Z 155.069,A -85,B 0,C 180,E1 -657.867,E2 -657.867} C_VEL
LIN {X 0,Y 601.444,Z 155.07,A -85,B 0,C 180,E1 -660.163,E2 -660.163} C_VEL
LIN {X 0,Y 601.417,Z 155.065,A -85,B 0,C 180,E1 -662.716,E2 -662.716} C_VEL
LIN {X 0,Y 601.413,Z 155.065,A -85,B 0,C 180,E1 -665.115,E2 -665.115} C_VEL
LIN {X 0,Y 601.429,Z 155.066,A -85,B 0,C 180,E1 -667.419,E2 -667.419} C_VEL
LIN {X 0,Y 601.409,Z 155.072,A -85,B 0,C 180,E1 -669.994,E2 -669.994} C_VEL
LIN {X 0,Y 601.405,Z 155.066,A -85,B 0,C 180,E1 -672.67,E2 -672.67} C_VEL
LIN {X 0,Y 601.419,Z 155.071,A -85,B 0,C 180,E1 -675.482,E2 -675.482} C_VEL
LIN {X 0,Y 601.419,Z 155.064,A -85,B 0,C 180,E1 -678.406,E2 -678.406} C_VEL
LIN {X 0,Y 601.427,Z 155.064,A -85,B 0,C 180,E1 -680.875,E2 -680.875} C_VEL
LIN {X 0,Y 601.438,Z 155.066,A -85,B 0,C 180,E1 -683.734,E2 -683.734} C_VEL
LIN {X 0,Y 601.426,Z 155.064,A -85,B 0,C 180,E1 -686.064,E2 -686.064} C_VEL
LIN {X 0,Y 601.422,Z 155.064,A -85,B 0,C 180,E1 -688.544,E2 -688.544} C_VEL
LIN {X 0,Y 601.431,Z 155.069,A -85,B 0,C 180,E1 -691.374,E2 -691.374} C_VEL
LIN {X 0,Y 601.397,Z 155.069,A -85,B 0,C 180,E1 -693.636,E2 -693.636} C_VEL
LIN {X 0,Y 601.413,Z 155.068,A -85,B 0,C 180,E1 -696.59,E2 -696.59} C_VEL
LIN {X 0,Y 601.429,Z 155.065,A -85,B 0,C 180,E1 -699.479,E2 -699.479} C_VEL
LIN {X 0,Y 601.391,Z 155.07,A -85,B 0,C 180,E1 -702.312,E2 -702.312} C_VEL
LIN {X 0,Y 601.409,Z 155.069,A -85,B 0,C 180,E1 -704.409,E2 -704.409} C_VEL
LIN {X 0,Y 601.424,Z 155.066,A -85,B 0,C 180,E1 -707.172,E2 -707.172} C_VEL
LIN {X 0,Y 601.421,Z 155.064,A -85,B 0,C 180,E1 -709.905,E2 -709.905} C_VEL
LIN {X 0,Y 601.448,Z 155.069,A -85,B 0,C 180,E1 -712.615,E2 -712.615} C_VEL
LIN {X 0,Y 601.416,Z 155.064,A -85,B 0,C 180,E1 -715.308,E2 -715.308} C_VEL
LIN {X 0,Y 601.412,Z 155.069,A -85,B 0,C 180,E1 -717.991,E2 -717.991} C_VEL
LIN {X 0,Y 601.453,Z 155.064,A -85,B 0,C 180,E1 -720.67,E2 -720.67} C_VEL
LIN {X 0,Y 601.415,Z 155.065,A -85,B 0,C 180,E1 -723.35,E2 -723.35} C_VEL
LIN {X 0,Y 601.406,Z 155.074,A -85,B 0,C 180,E1 -726.038,E2 -726.038} C_VEL
LIN {X 0,Y 601.434,Z 155.063,A -85,B 0,C 180,E1 -728.738,E2 -728.738} C_VEL
LIN {X 0,Y 601.405,Z 155.068,A -85,B 0,C 180,E1 -731.459,E2 -731.459} C_VEL
LIN {X 0,Y 601.415,Z 155.069,A -85,B 0,C 180,E1 -734.206,E2 -734.206} C_VEL
LIN {X 0,Y 601.422,Z 155.064,A -85,B 0,C 180,E1 -736.986,E2 -736.986} C_VEL
LIN {X 0,Y 601.399,Z 155.075,A -85,B 0,C 180,E1 -739.81,E2 -739.81} C_VEL
LIN {X 0,Y 601.405,Z 155.066,A -85,B 0,C 180,E1 -742.684,E2 -742.684} C_VEL
LIN {X 0,Y 601.393,Z 155.068,A -85,B 0,C 180,E1 -744.879,E2 -744.879} C_VEL
LIN {X 0,Y 601.407,Z 155.073,A -85,B 0,C 180,E1 -747.362,E2 -747.362} C_VEL
LIN {X 0,Y 601.424,Z 155.064,A -85,B 0,C 180,E1 -750.165,E2 -750.165} C_VEL
LIN {X 0,Y 601.403,Z 155.067,A -85,B 0,C 180,E1 -752.714,E2 -752.714} C_VEL
LIN {X 0,Y 601.385,Z 155.076,A -85,B 0,C 180,E1 -755.112,E2 -755.112} C_VEL
LIN {X 0,Y 601.432,Z 155.069,A -85,B 0,C 180,E1 -757.42,E2 -757.42} C_VEL
LIN {X 0,Y 601.409,Z 155.066,A -85,B 0,C 180,E1 -759.996,E2 -759.996} C_VEL
LIN {X 0,Y 601.384,Z 155.073,A -85,B 0,C 180,E1 -762.673,E2 -762.673} C_VEL
LIN {X 0,Y 601.396,Z 155.071,A -85,B 0,C 180,E1 -765.48,E2 -765.48} C_VEL
LIN {X 0,Y 601.415,Z 155.181,A -85,B 0,C 180,E1 -768.235,E2 -768.235} C_VEL
LIN {X 0,Y 601.453,Z 158.379,A -85,B 0,C 180,E1 -770.009,E2 -770.009} C_VEL
LIN {X 0,Y 601.445,Z 163.843,A -85,B 0,C 180,E1 -772.617,E2 -772.617} C_VEL
LIN {X 0,Y 601.458,Z 169.158,A -85,B 0,C 180,E1 -775.072,E2 -775.072} C_VEL
LIN {X 0,Y 601.444,Z 174.548,A -85,B 0,C 180,E1 -777.486,E2 -777.486} C_VEL
LIN {X 0,Y 601.43,Z 179.973,A -85,B 0,C 180,E1 -779.852,E2 -779.852} C_VEL
LIN {X 0,Y 601.406,Z 186.534,A -85,B 0,C 180,E1 -782.64,E2 -782.64} C_VEL
LIN {X 0,Y 601.399,Z 192.513,A -85,B 0,C 180,E1 -785.122,E2 -785.122} C_VEL
LIN {X 0,Y 601.386,Z 198.115,A -85,B 0,C 180,E1 -787.402,E2 -787.402} C_VEL
LIN {X 0,Y 601.369,Z 205.089,A -85,B 0,C 180,E1 -790.19,E2 -790.19} C_VEL
LIN {X 0,Y 601.346,Z 212.275,A -85,B 0,C 180,E1 -793.012,E2 -793.012} C_VEL
LIN {X 0,Y 601.306,Z 219.461,A -85,B 0,C 180,E1 -795.792,E2 -795.792} C_VEL
LIN {X 0,Y 601.354,Z 225.622,A -85,B 0,C 180,E1 -798.113,E2 -798.113} C_VEL
LIN {X 0,Y 601.611,Z 230.389,A -85,B 0,C 180,E1 -798.204,E2 -798.204} C_VEL
LIN {X 0,Y 601.572,Z 242.509,A -85,B 0,C 180,E1 -798.502,E2 -798.502} C_VEL
LIN {X 0,Y 601.481,Z 255.335,A -85,B 0,C 180,E1 -798.962,E2 -798.962} C_VEL
LIN {X 0,Y 601.457,Z 267.774,A -85,B 0,C 180,E1 -799.565,E2 -799.565} C_VEL
LIN {X 0,Y 601.467,Z 278.749,A -85,B 0,C 180,E1 -800.246,E2 -800.246} C_VEL
LIN {X 0,Y 601.435,Z 289.595,A -85,B 0,C 180,E1 -801.093,E2 -801.093} C_VEL
LIN {X 0,Y 601.406,Z 298.409,A -85,B 0,C 180,E1 -801.939,E2 -801.939} C_VEL
LIN {X 0,Y 601.377,Z 307.001,A -85,B 0,C 180,E1 -802.952,E2 -802.952} C_VEL
LIN {X 0,Y 601.36,Z 313.868,A -85,B 0,C 180,E1 -803.962,E2 -803.962} C_VEL
LIN {X 0,Y 601.345,Z 319.365,A -85,B 0,C 180,E1 -804.971,E2 -804.971} C_VEL
LIN {X 0,Y 601.347,Z 323.674,A -85,B 0,C 180,E1 -805.979,E2 -805.979} C_VEL
LIN {X 0,Y 601.344,Z 325.957,A -85,B 0,C 180,E1 -806.65,E2 -806.65} C_VEL
LIN {X 0,Y 601.325,Z 327.807,A -85,B 0,C 180,E1 -807.32,E2 -807.32} C_VEL
LIN {X 0,Y 601.343,Z 329.2,A -85,B 0,C 180,E1 -807.991,E2 -807.991} C_VEL
LIN {X 0,Y 601.339,Z 330.783,A -85,B 0,C 180,E1 -809.33,E2 -809.33} C_VEL
LIN {X 0,Y 601.335,Z 330.995,A -85,B 0,C 180,E1 -810,E2 -810} C_VEL
LIN {X 0,Y 601.347,Z 330.185,A -85,B 0,C 180,E1 -811.339,E2 -811.339} C_VEL
LIN {X 0,Y 601.343,Z 329.2,A -85,B 0,C 180,E1 -812.009,E2 -812.009} C_VEL
LIN {X 0,Y 601.325,Z 327.807,A -85,B 0,C 180,E1 -812.68,E2 -812.68} C_VEL
LIN {X 0,Y 601.368,Z 324.896,A -85,B 0,C 180,E1 -813.685,E2 -813.685} C_VEL
LIN {X 0,Y 601.336,Z 320.951,A -85,B 0,C 180,E1 -814.693,E2 -814.693} C_VEL
LIN {X 0,Y 601.372,Z 315.862,A -85,B 0,C 180,E1 -815.701,E2 -815.701} C_VEL
LIN {X 0,Y 601.382,Z 309.472,A -85,B 0,C 180,E1 -816.711,E2 -816.711} C_VEL
LIN {X 0,Y 601.396,Z 301.481,A -85,B 0,C 180,E1 -817.723,E2 -817.723} C_VEL
LIN {X 0,Y 601.423,Z 293.34,A -85,B 0,C 180,E1 -818.568,E2 -818.568} C_VEL
LIN {X 0,Y 601.455,Z 283.396,A -85,B 0,C 180,E1 -819.415,E2 -819.415} C_VEL
LIN {X 0,Y 601.447,Z 272.17,A -85,B 0,C 180,E1 -820.18,E2 -820.18} C_VEL
LIN {X 0,Y 601.451,Z 261.178,A -85,B 0,C 180,E1 -820.775,E2 -820.775} C_VEL
LIN {X 0,Y 601.531,Z 248.774,A -85,B 0,C 180,E1 -821.293,E2 -821.293} C_VEL
LIN {X 0,Y 601.585,Z 236.181,A -85,B 0,C 180,E1 -821.669,E2 -821.669} C_VEL
LIN {X 0,Y 601.426,Z 226.297,A -85,B 0,C 180,E1 -821.875,E2 -821.875} C_VEL
LIN {X 0,Y 601.327,Z 225.468,A -85,B 0,C 180,E1 -821.909,E2 -821.909} C_VEL
LIN {X 0,Y 601.335,Z 217.664,A -85,B 0,C 180,E1 -824.899,E2 -824.899} C_VEL
LIN {X 0,Y 601.367,Z 210.478,A -85,B 0,C 180,E1 -827.689,E2 -827.689} C_VEL
LIN {X 0,Y 601.374,Z 203.292,A -85,B 0,C 180,E1 -830.523,E2 -830.523} C_VEL
LIN {X 0,Y 601.384,Z 196.106,A -85,B 0,C 180,E1 -833.411,E2 -833.411} C_VEL
LIN {X 0,Y 601.392,Z 190.128,A -85,B 0,C 180,E1 -835.863,E2 -835.863} C_VEL
LIN {X 0,Y 601.427,Z 183.154,A -85,B 0,C 180,E1 -838.787,E2 -838.787} C_VEL
LIN {X 0,Y 601.442,Z 176.954,A -85,B 0,C 180,E1 -841.457,E2 -841.457} C_VEL
LIN {X 0,Y 601.428,Z 170.955,A -85,B 0,C 180,E1 -844.118,E2 -844.118} C_VEL
LIN {X 0,Y 601.445,Z 165.565,A -85,B 0,C 180,E1 -846.579,E2 -846.579} C_VEL
LIN {X 0,Y 601.465,Z 160.176,A -85,B 0,C 180,E1 -849.122,E2 -849.122} C_VEL
LIN {X 0,Y 601.512,Z 156.742,A -85,B 0,C 180,E1 -850.866,E2 -850.866} C_VEL
LIN {X 0,Y 601.415,Z 155.182,A -85,B 0,C 180,E1 -851.765,E2 -851.765} C_VEL
LIN {X 0,Y 601.423,Z 155.067,A -85,B 0,C 180,E1 -854.535,E2 -854.535} C_VEL
LIN {X 0,Y 601.384,Z 155.073,A -85,B 0,C 180,E1 -857.327,E2 -857.327} C_VEL
LIN {X 0,Y 601.409,Z 155.066,A -85,B 0,C 180,E1 -860.004,E2 -860.004} C_VEL
LIN {X 0,Y 601.433,Z 155.07,A -85,B 0,C 180,E1 -862.617,E2 -862.617} C_VEL
LIN {X 0,Y 601.394,Z 155.072,A -85,B 0,C 180,E1 -865.066,E2 -865.066} C_VEL
LIN {X 0,Y 601.405,Z 155.066,A -85,B 0,C 180,E1 -867.482,E2 -867.482} C_VEL
LIN {X 0,Y 601.425,Z 155.064,A -85,B 0,C 180,E1 -869.851,E2 -869.851} C_VEL
LIN {X 0,Y 601.436,Z 155.066,A -85,B 0,C 180,E1 -872.888,E2 -872.888} C_VEL
LIN {X 0,Y 601.46,Z 155.061,A -85,B 0,C 180,E1 -875.859,E2 -875.859} C_VEL
LIN {X 0,Y 601.398,Z 155.07,A -85,B 0,C 180,E1 -878.76,E2 -878.76} C_VEL
LIN {X 0,Y 601.418,Z 155.065,A -85,B 0,C 180,E1 -881.608,E2 -881.608} C_VEL
LIN {X 0,Y 601.44,Z 155.064,A -85,B 0,C 180,E1 -883.713,E2 -883.713} C_VEL
LIN {X 0,Y 601.405,Z 155.07,A -85,B 0,C 180,E1 -886.484,E2 -886.484} C_VEL
LIN {X 0,Y 601.415,Z 155.065,A -85,B 0,C 180,E1 -889.224,E2 -889.224} C_VEL
LIN {X 0,Y 601.436,Z 155.072,A -85,B 0,C 180,E1 -891.939,E2 -891.939} C_VEL
LIN {X 0,Y 601.412,Z 155.065,A -85,B 0,C 180,E1 -894.635,E2 -894.635} C_VEL
LIN {X 0,Y 601.443,Z 155.064,A -85,B 0,C 180,E1 -897.321,E2 -897.321} C_VEL
LIN {X 0,Y 601.433,Z 155.067,A -85,B 0,C 180,E1 -900,E2 -900} C_VEL
LIN {X 0,Y 601.433,Z 155.062,A -85,B 0,C 180,E1 -902.679,E2 -902.679} C_VEL
LIN {X 0,Y 601.427,Z 155.07,A -85,B 0,C 180,E1 -905.364,E2 -905.364} C_VEL
LIN {X 0,Y 601.428,Z 155.064,A -85,B 0,C 180,E1 -908.061,E2 -908.061} C_VEL
LIN {X 0,Y 601.424,Z 155.068,A -85,B 0,C 180,E1 -911.016,E2 -911.016} C_VEL
LIN {X 0,Y 601.403,Z 155.066,A -85,B 0,C 180,E1 -912.374,E2 -912.374} C_VEL
LIN {X 0,Y 600.746,Z 155.153,A -85,B 0,C 180,E1 -912.933,E2 -912.933} C_VEL
LIN {X 0,Y 597.899,Z 155.509,A -85,B 0,C 180,E1 -913.841,E2 -913.841} C_VEL
LIN {X 0,Y 595.486,Z 155.811,A -85,B 0,C 180,E1 -914.571,E2 -914.571} C_VEL
LIN {X 0,Y 594.445,Z 155.941,A -85,B 0,C 180,E1 -915.135,E2 -915.135} C_VEL
LIN {X 0,Y 594.358,Z 155.948,A -85,B 0,C 180,E1 -915.326,E2 -915.326} C_VEL
LIN {X 0,Y 594.385,Z 155.95,A -85,B 0,C 180,E1 -917.193,E2 -917.193} C_VEL
LIN {X 0,Y 594.371,Z 155.942,A -85,B 0,C 180,E1 -920.053,E2 -920.053} C_VEL
LIN {X 0,Y 594.357,Z 155.953,A -85,B 0,C 180,E1 -922.967,E2 -922.967} C_VEL
LIN {X 0,Y 594.368,Z 155.948,A -85,B 0,C 180,E1 -925.193,E2 -925.193} C_VEL
LIN {X 0,Y 594.378,Z 155.942,A -85,B 0,C 180,E1 -927.527,E2 -927.527} C_VEL
LIN {X 0,Y 594.393,Z 155.942,A -85,B 0,C 180,E1 -930.331,E2 -930.331} C_VEL
LIN {X 0,Y 594.372,Z 155.948,A -85,B 0,C 180,E1 -932.95,E2 -932.95} C_VEL
LIN {X 0,Y 594.376,Z 155.942,A -85,B 0,C 180,E1 -935.407,E2 -935.407} C_VEL
LIN {X 0,Y 594.381,Z 155.942,A -85,B 0,C 180,E1 -937.941,E2 -937.941} C_VEL
LIN {X 0,Y 594.38,Z 155.945,A -85,B 0,C 180,E1 -940.823,E2 -940.823} C_VEL
LIN {X 0,Y 594.375,Z 155.944,A -85,B 0,C 180,E1 -943.841,E2 -943.841} C_VEL
LIN {X 0,Y 594.36,Z 155.947,A -85,B 0,C 180,E1 -946.701,E2 -946.701} C_VEL
LIN {X 0,Y 594.367,Z 155.943,A -85,B 0,C 180,E1 -949.434,E2 -949.434} C_VEL
LIN {X 0,Y 594.384,Z 155.946,A -85,B 0,C 180,E1 -952.392,E2 -952.392} C_VEL
LIN {X 0,Y 594.381,Z 155.942,A -85,B 0,C 180,E1 -954.672,E2 -954.672} C_VEL
LIN {X 0,Y 594.374,Z 155.942,A -85,B 0,C 180,E1 -957.088,E2 -957.088} C_VEL
LIN {X 0,Y 594.396,Z 155.945,A -85,B 0,C 180,E1 -959.669,E2 -959.669} C_VEL
LIN {X 0,Y 594.369,Z 155.943,A -85,B 0,C 180,E1 -962.539,E2 -962.539} C_VEL
LIN {X 0,Y 594.371,Z 155.942,A -85,B 0,C 180,E1 -964.807,E2 -964.807} C_VEL
LIN {X 0,Y 594.36,Z 155.947,A -85,B 0,C 180,E1 -967.265,E2 -967.265} C_VEL
LIN {X 0,Y 594.373,Z 155.946,A -85,B 0,C 180,E1 -969.947,E2 -969.947} C_VEL
LIN {X 0,Y 594.388,Z 155.941,A -85,B 0,C 180,E1 -972.807,E2 -972.807} C_VEL
LIN {X 0,Y 594.385,Z 155.944,A -85,B 0,C 180,E1 -975.826,E2 -975.826} C_VEL
LIN {X 0,Y 594.391,Z 155.94,A -85,B 0,C 180,E1 -978.404,E2 -978.404} C_VEL
LIN {X 0,Y 594.395,Z 155.948,A -85,B 0,C 180,E1 -981.158,E2 -981.158} C_VEL
LIN {X 0,Y 594.391,Z 155.941,A -85,B 0,C 180,E1 -983.891,E2 -983.891} C_VEL
LIN {X 0,Y 594.375,Z 155.945,A -85,B 0,C 180,E1 -986.611,E2 -986.611} C_VEL
LIN {X 0,Y 594.418,Z 155.942,A -85,B 0,C 180,E1 -989.323,E2 -989.323} C_VEL
LIN {X 0,Y 594.404,Z 155.938,A -85,B 0,C 180,E1 -992.033,E2 -992.033} C_VEL
LIN {X 0,Y 594.389,Z 155.949,A -85,B 0,C 180,E1 -994.748,E2 -994.748} C_VEL
LIN {X 0,Y 594.39,Z 155.941,A -85,B 0,C 180,E1 -997.473,E2 -997.473} C_VEL
LIN {X 0,Y 594.393,Z 155.942,A -85,B 0,C 180,E1 -1000.216,E2 -1000.216} C_VEL
LIN {X 0,Y 594.367,Z 155.947,A -85,B 0,C 180,E1 -1002.983,E2 -1002.983} C_VEL
LIN {X 0,Y 594.364,Z 155.944,A -85,B 0,C 180,E1 -1005.781,E2 -1005.781} C_VEL
LIN {X 0,Y 594.384,Z 155.948,A -85,B 0,C 180,E1 -1008.617,E2 -1008.617} C_VEL
LIN {X 0,Y 594.365,Z 155.943,A -85,B 0,C 180,E1 -1011.503,E2 -1011.503} C_VEL
LIN {X 0,Y 594.385,Z 155.947,A -85,B 0,C 180,E1 -1014.446,E2 -1014.446} C_VEL
LIN {X 0,Y 594.385,Z 155.943,A -85,B 0,C 180,E1 -1016.699,E2 -1016.699} C_VEL
LIN {X 0,Y 594.377,Z 155.941,A -85,B 0,C 180,E1 -1018.998,E2 -1018.998} C_VEL
LIN {X 0,Y 594.387,Z 155.944,A -85,B 0,C 180,E1 -1021.645,E2 -1021.645} C_VEL
LIN {X 0,Y 594.395,Z 155.94,A -85,B 0,C 180,E1 -1024.578,E2 -1024.578} C_VEL
LIN {X 0,Y 594.38,Z 155.941,A -85,B 0,C 180,E1 -1027.086,E2 -1027.086} C_VEL
LIN {X 0,Y 594.373,Z 155.951,A -85,B 0,C 180,E1 -1029.775,E2 -1029.775} C_VEL
LIN {X 0,Y 594.364,Z 155.944,A -85,B 0,C 180,E1 -1032.375,E2 -1032.375} C_VEL
LIN {X 0,Y 594.356,Z 155.947,A -85,B 0,C 180,E1 -1035.191,E2 -1035.191} C_VEL
LIN {X 0,Y 594.366,Z 155.952,A -85,B 0,C 180,E1 -1037.625,E2 -1037.625} C_VEL
LIN {X 0,Y 594.387,Z 155.94,A -85,B 0,C 180,E1 -1040.321,E2 -1040.321} C_VEL
LIN {X 0,Y 594.378,Z 155.944,A -85,B 0,C 180,E1 -1042.913,E2 -1042.913} C_VEL
LIN {X 0,Y 594.379,Z 155.943,A -85,B 0,C 180,E1 -1045.86,E2 -1045.86} C_VEL
LIN {X 0,Y 594.373,Z 155.943,A -85,B 0,C 180,E1 -1048.65,E2 -1048.65} C_VEL
LIN {X 0,Y 594.378,Z 155.949,A -85,B 0,C 180,E1 -1051.042,E2 -1051.042} C_VEL
LIN {X 0,Y 594.376,Z 155.941,A -85,B 0,C 180,E1 -1053.978,E2 -1053.978} C_VEL
LIN {X 0,Y 594.385,Z 155.941,A -85,B 0,C 180,E1 -1056.296,E2 -1056.296} C_VEL
LIN {X 0,Y 594.402,Z 155.943,A -85,B 0,C 180,E1 -1059.225,E2 -1059.225} C_VEL
LIN {X 0,Y 594.348,Z 155.945,A -85,B 0,C 180,E1 -1062.095,E2 -1062.095} C_VEL
LIN {X 0,Y 594.362,Z 155.945,A -85,B 0,C 180,E1 -1064.219,E2 -1064.219} C_VEL
LIN {X 0,Y 594.369,Z 155.947,A -85,B 0,C 180,E1 -1067.017,E2 -1067.017} C_VEL
LIN {X 0,Y 594.383,Z 155.941,A -85,B 0,C 180,E1 -1069.784,E2 -1069.784} C_VEL
LIN {X 0,Y 594.396,Z 155.949,A -85,B 0,C 180,E1 -1072.527,E2 -1072.527} C_VEL
LIN {X 0,Y 594.386,Z 155.94,A -85,B 0,C 180,E1 -1075.253,E2 -1075.253} C_VEL
LIN {X 0,Y 594.383,Z 155.944,A -85,B 0,C 180,E1 -1077.968,E2 -1077.968} C_VEL
LIN {X 0,Y 594.423,Z 155.939,A -85,B 0,C 180,E1 -1080.678,E2 -1080.678} C_VEL
LIN {X 0,Y 594.367,Z 155.943,A -85,B 0,C 180,E1 -1083.39,E2 -1083.39} C_VEL
LIN {X 0,Y 594.36,Z 155.953,A -85,B 0,C 180,E1 -1086.109,E2 -1086.109} C_VEL
LIN {X 0,Y 594.393,Z 155.94,A -85,B 0,C 180,E1 -1088.842,E2 -1088.842} C_VEL
LIN {X 0,Y 594.374,Z 155.946,A -85,B 0,C 180,E1 -1091.596,E2 -1091.596} C_VEL
LIN {X 0,Y 594.384,Z 155.943,A -85,B 0,C 180,E1 -1094.378,E2 -1094.378} C_VEL
LIN {X 0,Y 594.381,Z 155.942,A -85,B 0,C 180,E1 -1097.194,E2 -1097.194} C_VEL
LIN {X 0,Y 594.368,Z 155.947,A -85,B 0,C 180,E1 -1100.054,E2 -1100.054} C_VEL
LIN {X 0,Y 594.358,Z 155.945,A -85,B 0,C 180,E1 -1102.968,E2 -1102.968} C_VEL
LIN {X 0,Y 594.372,Z 155.946,A -85,B 0,C 180,E1 -1105.194,E2 -1105.194} C_VEL
LIN {X 0,Y 594.381,Z 155.95,A -85,B 0,C 180,E1 -1107.527,E2 -1107.527} C_VEL
LIN {X 0,Y 594.378,Z 155.941,A -85,B 0,C 180,E1 -1110.56,E2 -1110.56} C_VEL
LIN {X 0,Y 594.372,Z 155.946,A -85,B 0,C 180,E1 -1112.951,E2 -1112.951} C_VEL
LIN {X 0,Y 594.345,Z 155.953,A -85,B 0,C 180,E1 -1115.41,E2 -1115.41} C_VEL
LIN {X 0,Y 594.376,Z 155.942,A -85,B 0,C 180,E1 -1117.942,E2 -1117.942} C_VEL
LIN {X 0,Y 594.371,Z 155.948,A -85,B 0,C 180,E1 -1120.822,E2 -1120.822} C_VEL
LIN {X 0,Y 594.357,Z 155.945,A -85,B 0,C 180,E1 -1123.839,E2 -1123.839} C_VEL
LIN {X 0,Y 594.35,Z 155.953,A -85,B 0,C 180,E1 -1126.7,E2 -1126.7} C_VEL
LIN {X 0,Y 594.364,Z 155.95,A -85,B 0,C 180,E1 -1127.625,E2 -1127.625} C_VEL
LIN {X 0,Y 594.496,Z 157.037,A -85,B 0,C 180,E1 -1128.547,E2 -1128.547} C_VEL
LIN {X 0,Y 594.469,Z 162.145,A -85,B 0,C 180,E1 -1131.286,E2 -1131.286} C_VEL
LIN {X 0,Y 594.417,Z 167.362,A -85,B 0,C 180,E1 -1133.761,E2 -1133.761} C_VEL
LIN {X 0,Y 594.394,Z 172.751,A -85,B 0,C 180,E1 -1136.24,E2 -1136.24} C_VEL
LIN {X 0,Y 594.394,Z 178.141,A -85,B 0,C 180,E1 -1138.652,E2 -1138.652} C_VEL
LIN {X 0,Y 594.38,Z 183.627,A -85,B 0,C 180,E1 -1141.043,E2 -1141.043} C_VEL
LIN {X 0,Y 594.344,Z 188.92,A -85,B 0,C 180,E1 -1143.299,E2 -1143.299} C_VEL
LIN {X 0,Y 594.336,Z 194.373,A -85,B 0,C 180,E1 -1145.578,E2 -1145.578} C_VEL
LIN {X 0,Y 594.316,Z 199.699,A -85,B 0,C 180,E1 -1147.765,E2 -1147.765} C_VEL
LIN {X 0,Y 594.287,Z 205.089,A -85,B 0,C 180,E1 -1149.944,E2 -1149.944} C_VEL
LIN {X 0,Y 594.275,Z 210.478,A -85,B 0,C 180,E1 -1152.093,E2 -1152.093} C_VEL
LIN {X 0,Y 594.262,Z 217.664,A -85,B 0,C 180,E1 -1154.919,E2 -1154.919} C_VEL
LIN {X 0,Y 594.263,Z 225.603,A -85,B 0,C 180,E1 -1157.969,E2 -1157.969} C_VEL
LIN {X 0,Y 594.66,Z 231.53,A -85,B 0,C 180,E1 -1158.086,E2 -1158.086} C_VEL
LIN {X 0,Y 594.615,Z 243.863,A -85,B 0,C 180,E1 -1158.409,E2 -1158.409} C_VEL
LIN {X 0,Y 594.519,Z 256.094,A -85,B 0,C 180,E1 -1158.865,E2 -1158.865} C_VEL
LIN {X 0,Y 594.473,Z 267.774,A -85,B 0,C 180,E1 -1159.441,E2 -1159.441} C_VEL
LIN {X 0,Y 594.446,Z 278.75,A -85,B 0,C 180,E1 -1160.129,E2 -1160.129} C_VEL
LIN {X 0,Y 594.404,Z 289.593,A -85,B 0,C 180,E1 -1160.987,E2 -1160.987} C_VEL
LIN {X 0,Y 594.365,Z 298.406,A -85,B 0,C 180,E1 -1161.843,E2 -1161.843} C_VEL
LIN {X 0,Y 594.304,Z 307.002,A -85,B 0,C 180,E1 -1162.867,E2 -1162.867} C_VEL
LIN {X 0,Y 594.289,Z 313.868,A -85,B 0,C 180,E1 -1163.89,E2 -1163.89} C_VEL
LIN {X 0,Y 594.254,Z 319.365,A -85,B 0,C 180,E1 -1164.911,E2 -1164.911} C_VEL
LIN {X 0,Y 594.262,Z 323.672,A -85,B 0,C 180,E1 -1165.931,E2 -1165.931} C_VEL
LIN {X 0,Y 594.267,Z 325.959,A -85,B 0,C 180,E1 -1166.61,E2 -1166.61} C_VEL
LIN {X 0,Y 594.226,Z 327.805,A -85,B 0,C 180,E1 -1167.288,E2 -1167.288} C_VEL
LIN {X 0,Y 594.242,Z 329.199,A -85,B 0,C 180,E1 -1167.967,E2 -1167.967} C_VEL
LIN {X 0,Y 594.239,Z 330.783,A -85,B 0,C 180,E1 -1169.322,E2 -1169.322} C_VEL
LIN {X 0,Y 594.236,Z 330.991,A -85,B 0,C 180,E1 -1170,E2 -1170} C_VEL
LIN {X 0,Y 594.247,Z 330.186,A -85,B 0,C 180,E1 -1171.355,E2 -1171.355} C_VEL
LIN {X 0,Y 594.242,Z 329.199,A -85,B 0,C 180,E1 -1172.033,E2 -1172.033} C_VEL
LIN {X 0,Y 594.226,Z 327.805,A -85,B 0,C 180,E1 -1172.712,E2 -1172.712} C_VEL
LIN {X 0,Y 594.289,Z 324.894,A -85,B 0,C 180,E1 -1173.729,E2 -1173.729} C_VEL
LIN {X 0,Y 594.241,Z 320.949,A -85,B 0,C 180,E1 -1174.749,E2 -1174.749} C_VEL
LIN {X 0,Y 594.299,Z 315.858,A -85,B 0,C 180,E1 -1175.769,E2 -1175.769} C_VEL
LIN {X 0,Y 594.316,Z 309.471,A -85,B 0,C 180,E1 -1176.791,E2 -1176.791} C_VEL
LIN {X 0,Y 594.346,Z 301.482,A -85,B 0,C 180,E1 -1177.815,E2 -1177.815} C_VEL
LIN {X 0,Y 594.377,Z 293.342,A -85,B 0,C 180,E1 -1178.671,E2 -1178.671} C_VEL
LIN {X 0,Y 594.419,Z 283.39,A -85,B 0,C 180,E1 -1179.528,E2 -1179.528} C_VEL
LIN {X 0,Y 594.431,Z 273.577,A -85,B 0,C 180,E1 -1180.215,E2 -1180.215} C_VEL
LIN {X 0,Y 594.476,Z 261.181,A -85,B 0,C 180,E1 -1180.903,E2 -1180.903} C_VEL
LIN {X 0,Y 594.565,Z 249.055,A -85,B 0,C 180,E1 -1181.417,E2 -1181.417} C_VEL
LIN {X 0,Y 594.655,Z 236.176,A -85,B 0,C 180,E1 -1181.806,E2 -1181.806} C_VEL
LIN {X 0,Y 594.529,Z 227.248,A -85,B 0,C 180,E1 -1181.998,E2 -1181.998} C_VEL
LIN {X 0,Y 594.266,Z 225.468,A -85,B 0,C 180,E1 -1182.052,E2 -1182.052} C_VEL
LIN {X 0,Y 594.262,Z 217.664,A -85,B 0,C 180,E1 -1185.081,E2 -1185.081} C_VEL
LIN {X 0,Y 594.275,Z 210.478,A -85,B 0,C 180,E1 -1187.907,E2 -1187.907} C_VEL
LIN {X 0,Y 594.323,Z 202.987,A -85,B 0,C 180,E1 -1190.901,E2 -1190.901} C_VEL
LIN {X 0,Y 594.309,Z 196.106,A -85,B 0,C 180,E1 -1193.707,E2 -1193.707} C_VEL
LIN {X 0,Y 594.332,Z 190.56,A -85,B 0,C 180,E1 -1196.011,E2 -1196.011} C_VEL
LIN {X 0,Y 594.34,Z 185.327,A -85,B 0,C 180,E1 -1198.228,E2 -1198.228} C_VEL
LIN {X 0,Y 594.389,Z 179.937,A -85,B 0,C 180,E1 -1200.559,E2 -1200.559} C_VEL
LIN {X 0,Y 594.423,Z 174.548,A -85,B 0,C 180,E1 -1202.947,E2 -1202.947} C_VEL
LIN {X 0,Y 594.444,Z 169.158,A -85,B 0,C 180,E1 -1205.402,E2 -1205.402} C_VEL
LIN {X 0,Y 594.434,Z 163.769,A -85,B 0,C 180,E1 -1207.936,E2 -1207.936} C_VEL
LIN {X 0,Y 594.541,Z 158.108,A -85,B 0,C 180,E1 -1210.84,E2 -1210.84} C_VEL
LIN {X 0,Y 594.414,Z 156.39,A -85,B 0,C 180,E1 -1211.851,E2 -1211.851} C_VEL
LIN {X 0,Y 594.364,Z 155.95,A -85,B 0,C 180,E1 -1212.375,E2 -1212.375} C_VEL
LIN {X 0,Y 594.343,Z 155.954,A -85,B 0,C 180,E1 -1215.192,E2 -1215.192} C_VEL
LIN {X 0,Y 594.372,Z 155.943,A -85,B 0,C 180,E1 -1218.152,E2 -1218.152} C_VEL
LIN {X 0,Y 594.376,Z 155.946,A -85,B 0,C 180,E1 -1221.194,E2 -1221.194} C_VEL
LIN {X 0,Y 594.345,Z 155.945,A -85,B 0,C 180,E1 -1223.755,E2 -1223.755} C_VEL
LIN {X 0,Y 594.376,Z 155.944,A -85,B 0,C 180,E1 -1226.238,E2 -1226.238} C_VEL
LIN {X 0,Y 594.374,Z 155.951,A -85,B 0,C 180,E1 -1228.65,E2 -1228.65} C_VEL
LIN {X 0,Y 594.372,Z 155.944,A -85,B 0,C 180,E1 -1231.043,E2 -1231.043} C_VEL
LIN {X 0,Y 594.373,Z 155.942,A -85,B 0,C 180,E1 -1233.3,E2 -1233.3} C_VEL
LIN {X 0,Y 594.387,Z 155.948,A -85,B 0,C 180,E1 -1236.296,E2 -1236.296} C_VEL
LIN {X 0,Y 594.394,Z 155.939,A -85,B 0,C 180,E1 -1239.224,E2 -1239.224} C_VEL
LIN {X 0,Y 594.348,Z 155.953,A -85,B 0,C 180,E1 -1242.094,E2 -1242.094} C_VEL
LIN {X 0,Y 594.36,Z 155.953,A -85,B 0,C 180,E1 -1244.219,E2 -1244.219} C_VEL
LIN {X 0,Y 594.372,Z 155.948,A -85,B 0,C 180,E1 -1246.32,E2 -1246.32} C_VEL
LIN {X 0,Y 594.373,Z 155.942,A -85,B 0,C 180,E1 -1249.094,E2 -1249.094} C_VEL
LIN {X 0,Y 594.412,Z 155.946,A -85,B 0,C 180,E1 -1251.843,E2 -1251.843} C_VEL
LIN {X 0,Y 594.378,Z 155.942,A -85,B 0,C 180,E1 -1254.572,E2 -1254.572} C_VEL
LIN {X 0,Y 594.407,Z 155.94,A -85,B 0,C 180,E1 -1257.289,E2 -1257.289} C_VEL
LIN {X 0,Y 594.402,Z 155.943,A -85,B 0,C 180,E1 -1260,E2 -1260} C_VEL
LIN {X 0,Y 594.399,Z 155.938,A -85,B 0,C 180,E1 -1262.71,E2 -1262.71} C_VEL
LIN {X 0,Y 594.39,Z 155.948,A -85,B 0,C 180,E1 -1265.427,E2 -1265.427} C_VEL
LIN {X 0,Y 594.406,Z 155.938,A -85,B 0,C 180,E1 -1268.156,E2 -1268.156} C_VEL
LIN {X 0,Y 594.388,Z 155.945,A -85,B 0,C 180,E1 -1271.077,E2 -1271.077} C_VEL
LIN {X 0,Y 594.376,Z 155.945,A -85,B 0,C 180,E1 -1273.679,E2 -1273.679} C_VEL
LIN {X 0,Y 594.358,Z 155.948,A -85,B 0,C 180,E1 -1275.326,E2 -1275.326} C_VEL
LIN {X 0,Y 593.682,Z 156.03,A -85,B 0,C 180,E1 -1275.891,E2 -1275.891} C_VEL
LIN {X 0,Y 590.814,Z 156.389,A -85,B 0,C 180,E1 -1276.809,E2 -1276.809} C_VEL
LIN {X 0,Y 588.405,Z 156.689,A -85,B 0,C 180,E1 -1277.548,E2 -1277.548} C_VEL
LIN {X 0,Y 587.382,Z 156.813,A -85,B 0,C 180,E1 -1278.118,E2 -1278.118} C_VEL
LIN {X 0,Y 587.306,Z 156.822,A -85,B 0,C 180,E1 -1278.311,E2 -1278.311} C_VEL
LIN {X 0,Y 587.351,Z 156.827,A -85,B 0,C 180,E1 -1281.045,E2 -1281.045} C_VEL
LIN {X 0,Y 587.331,Z 156.819,A -85,B 0,C 180,E1 -1284.006,E2 -1284.006} C_VEL
LIN {X 0,Y 587.331,Z 156.82,A -85,B 0,C 180,E1 -1286.278,E2 -1286.278} C_VEL
LIN {X 0,Y 587.344,Z 156.822,A -85,B 0,C 180,E1 -1289.134,E2 -1289.134} C_VEL
LIN {X 0,Y 587.343,Z 156.817,A -85,B 0,C 180,E1 -1291.837,E2 -1291.837} C_VEL
LIN {X 0,Y 587.35,Z 156.821,A -85,B 0,C 180,E1 -1294.349,E2 -1294.349} C_VEL
LIN {X 0,Y 587.346,Z 156.824,A -85,B 0,C 180,E1 -1296.747,E2 -1296.747} C_VEL
LIN {X 0,Y 587.34,Z 156.818,A -85,B 0,C 180,E1 -1299.359,E2 -1299.359} C_VEL
LIN {X 0,Y 587.328,Z 156.824,A -85,B 0,C 180,E1 -1302.108,E2 -1302.108} C_VEL
LIN {X 0,Y 587.309,Z 156.822,A -85,B 0,C 180,E1 -1305.089,E2 -1305.089} C_VEL
LIN {X 0,Y 587.347,Z 156.822,A -85,B 0,C 180,E1 -1307.928,E2 -1307.928} C_VEL
LIN {X 0,Y 587.328,Z 156.819,A -85,B 0,C 180,E1 -1311.058,E2 -1311.058} C_VEL
LIN {X 0,Y 587.349,Z 156.817,A -85,B 0,C 180,E1 -1313.292,E2 -1313.292} C_VEL
LIN {X 0,Y 587.364,Z 156.821,A -85,B 0,C 180,E1 -1315.781,E2 -1315.781} C_VEL
LIN {X 0,Y 587.348,Z 156.822,A -85,B 0,C 180,E1 -1318.232,E2 -1318.232} C_VEL
LIN {X 0,Y 587.346,Z 156.817,A -85,B 0,C 180,E1 -1320.866,E2 -1320.866} C_VEL
LIN {X 0,Y 587.354,Z 156.826,A -85,B 0,C 180,E1 -1323.819,E2 -1323.819} C_VEL
LIN {X 0,Y 587.333,Z 156.824,A -85,B 0,C 180,E1 -1325.994,E2 -1325.994} C_VEL
LIN {X 0,Y 587.32,Z 156.822,A -85,B 0,C 180,E1 -1328.226,E2 -1328.226} C_VEL
LIN {X 0,Y 587.348,Z 156.82,A -85,B 0,C 180,E1 -1331.151,E2 -1331.151} C_VEL
LIN {X 0,Y 587.322,Z 156.823,A -85,B 0,C 180,E1 -1334.025,E2 -1334.025} C_VEL
LIN {X 0,Y 587.356,Z 156.817,A -85,B 0,C 180,E1 -1336.154,E2 -1336.154} C_VEL
LIN {X 0,Y 587.341,Z 156.822,A -85,B 0,C 180,E1 -1338.963,E2 -1338.963} C_VEL
LIN {X 0,Y 587.368,Z 156.818,A -85,B 0,C 180,E1 -1341.745,E2 -1341.745} C_VEL
LIN {X 0,Y 587.361,Z 156.817,A -85,B 0,C 180,E1 -1344.507,E2 -1344.507} C_VEL
LIN {X 0,Y 587.37,Z 156.822,A -85,B 0,C 180,E1 -1347.257,E2 -1347.257} C_VEL
LIN {X 0,Y 587.382,Z 156.813,A -85,B 0,C 180,E1 -1350,E2 -1350} C_VEL
LIN {X 0,Y 587.37,Z 156.822,A -85,B 0,C 180,E1 -1352.743,E2 -1352.743} C_VEL
LIN {X 0,Y 587.361,Z 156.817,A -85,B 0,C 180,E1 -1355.493,E2 -1355.493} C_VEL
LIN {X 0,Y 587.368,Z 156.818,A -85,B 0,C 180,E1 -1358.255,E2 -1358.255} C_VEL
LIN {X 0,Y 587.345,Z 156.821,A -85,B 0,C 180,E1 -1361.134,E2 -1361.134} C_VEL
LIN {X 0,Y 587.361,Z 156.821,A -85,B 0,C 180,E1 -1364.26,E2 -1364.26} C_VEL
LIN {X 0,Y 587.348,Z 156.817,A -85,B 0,C 180,E1 -1367.406,E2 -1367.406} C_VEL
LIN {X 0,Y 587.329,Z 156.828,A -85,B 0,C 180,E1 -1370.305,E2 -1370.305} C_VEL
LIN {X 0,Y 587.318,Z 156.82,A -85,B 0,C 180,E1 -1373.258,E2 -1373.258} C_VEL
LIN {X 0,Y 587.329,Z 156.82,A -85,B 0,C 180,E1 -1375.516,E2 -1375.516} C_VEL
LIN {X 0,Y 587.345,Z 156.822,A -85,B 0,C 180,E1 -1377.817,E2 -1377.817} C_VEL
LIN {X 0,Y 587.347,Z 156.82,A -85,B 0,C 180,E1 -1380.512,E2 -1380.512} C_VEL
LIN {X 0,Y 587.33,Z 156.821,A -85,B 0,C 180,E1 -1383.396,E2 -1383.396} C_VEL
LIN {X 0,Y 587.352,Z 156.826,A -85,B 0,C 180,E1 -1385.895,E2 -1385.895} C_VEL
LIN {X 0,Y 587.328,Z 156.821,A -85,B 0,C 180,E1 -1388.479,E2 -1388.479} C_VEL
LIN {X 0,Y 587.333,Z 156.82,A -85,B 0,C 180,E1 -1391.156,E2 -1391.156} C_VEL
LIN {X 0,Y 587.32,Z 156.824,A -85,B 0,C 180,E1 -1394.113,E2 -1394.113} C_VEL
LIN {X 0,Y 587.315,Z 156.822,A -85,B 0,C 180,E1 -1396.994,E2 -1396.994} C_VEL
LIN {X 0,Y 587.314,Z 156.827,A -85,B 0,C 180,E1 -1399.746,E2 -1399.746} C_VEL
LIN {X 0,Y 587.338,Z 156.818,A -85,B 0,C 180,E1 -1402.392,E2 -1402.392} C_VEL
LIN {X 0,Y 587.344,Z 156.821,A -85,B 0,C 180,E1 -1404.946,E2 -1404.946} C_VEL
LIN {X 0,Y 587.333,Z 156.826,A -85,B 0,C 180,E1 -1407.421,E2 -1407.421} C_VEL
LIN {X 0,Y 587.339,Z 156.819,A -85,B 0,C 180,E1 -1409.831,E2 -1409.831} C_VEL
LIN {X 0,Y 587.344,Z 156.817,A -85,B 0,C 180,E1 -1412.307,E2 -1412.307} C_VEL
LIN {X 0,Y 587.344,Z 156.824,A -85,B 0,C 180,E1 -1415.242,E2 -1415.242} C_VEL
LIN {X 0,Y 587.315,Z 156.822,A -85,B 0,C 180,E1 -1418.226,E2 -1418.226} C_VEL
LIN {X 0,Y 587.346,Z 156.822,A -85,B 0,C 180,E1 -1421.152,E2 -1421.152} C_VEL
LIN {X 0,Y 587.32,Z 156.821,A -85,B 0,C 180,E1 -1424.025,E2 -1424.025} C_VEL
LIN {X 0,Y 587.353,Z 156.818,A -85,B 0,C 180,E1 -1426.155,E2 -1426.155} C_VEL
LIN {X 0,Y 587.339,Z 156.823,A -85,B 0,C 180,E1 -1428.963,E2 -1428.963} C_VEL
LIN {X 0,Y 587.361,Z 156.815,A -85,B 0,C 180,E1 -1431.745,E2 -1431.745} C_VEL
LIN {X 0,Y 587.353,Z 156.826,A -85,B 0,C 180,E1 -1434.507,E2 -1434.507} C_VEL
LIN {X 0,Y 587.366,Z 156.815,A -85,B 0,C 180,E1 -1437.257,E2 -1437.257} C_VEL
LIN {X 0,Y 587.372,Z 156.819,A -85,B 0,C 180,E1 -1440,E2 -1440} C_VEL
LIN {X 0,Y 587.372,Z 156.816,A -85,B 0,C 180,E1 -1442.744,E2 -1442.744} C_VEL
LIN {X 0,Y 587.344,Z 156.818,A -85,B 0,C 180,E1 -1445.493,E2 -1445.493} C_VEL
LIN {X 0,Y 587.366,Z 156.821,A -85,B 0,C 180,E1 -1448.256,E2 -1448.256} C_VEL
LIN {X 0,Y 587.342,Z 156.818,A -85,B 0,C 180,E1 -1451.134,E2 -1451.134} C_VEL
LIN {X 0,Y 587.36,Z 156.819,A -85,B 0,C 180,E1 -1454.261,E2 -1454.261} C_VEL
LIN {X 0,Y 587.343,Z 156.821,A -85,B 0,C 180,E1 -1457.407,E2 -1457.407} C_VEL
LIN {X 0,Y 587.322,Z 156.822,A -85,B 0,C 180,E1 -1460.305,E2 -1460.305} C_VEL
LIN {X 0,Y 587.318,Z 156.825,A -85,B 0,C 180,E1 -1463.259,E2 -1463.259} C_VEL
LIN {X 0,Y 587.333,Z 156.828,A -85,B 0,C 180,E1 -1465.517,E2 -1465.517} C_VEL
LIN {X 0,Y 587.34,Z 156.822,A -85,B 0,C 180,E1 -1467.818,E2 -1467.818} C_VEL
LIN {X 0,Y 587.333,Z 156.819,A -85,B 0,C 180,E1 -1470.511,E2 -1470.511} C_VEL
LIN {X 0,Y 587.33,Z 156.828,A -85,B 0,C 180,E1 -1473.397,E2 -1473.397} C_VEL
LIN {X 0,Y 587.286,Z 156.826,A -85,B 0,C 180,E1 -1475.901,E2 -1475.901} C_VEL
LIN {X 0,Y 587.32,Z 156.822,A -85,B 0,C 180,E1 -1478.48,E2 -1478.48} C_VEL
LIN {X 0,Y 587.333,Z 156.829,A -85,B 0,C 180,E1 -1481.158,E2 -1481.158} C_VEL
LIN {X 0,Y 587.309,Z 156.824,A -85,B 0,C 180,E1 -1484.112,E2 -1484.112} C_VEL
LIN {X 0,Y 587.305,Z 156.832,A -85,B 0,C 180,E1 -1486.994,E2 -1486.994} C_VEL
LIN {X 0,Y 587.388,Z 157.38,A -85,B 0,C 180,E1 -1487.931,E2 -1487.931} C_VEL
LIN {X 0,Y 587.515,Z 160.523,A -85,B 0,C 180,E1 -1489.763,E2 -1489.763} C_VEL
LIN {X 0,Y 587.407,Z 165.565,A -85,B 0,C 180,E1 -1492.398,E2 -1492.398} C_VEL
LIN {X 0,Y 587.39,Z 170.955,A -85,B 0,C 180,E1 -1494.949,E2 -1494.949} C_VEL
LIN {X 0,Y 587.367,Z 176.344,A -85,B 0,C 180,E1 -1497.423,E2 -1497.423} C_VEL
LIN {X 0,Y 587.334,Z 181.734,A -85,B 0,C 180,E1 -1499.83,E2 -1499.83} C_VEL
LIN {X 0,Y 587.298,Z 187.442,A -85,B 0,C 180,E1 -1502.318,E2 -1502.318} C_VEL
LIN {X 0,Y 587.293,Z 194.309,A -85,B 0,C 180,E1 -1505.239,E2 -1505.239} C_VEL
LIN {X 0,Y 587.247,Z 201.495,A -85,B 0,C 180,E1 -1508.223,E2 -1508.223} C_VEL
LIN {X 0,Y 587.241,Z 208.682,A -85,B 0,C 180,E1 -1511.148,E2 -1511.148} C_VEL
LIN {X 0,Y 587.183,Z 215.868,A -85,B 0,C 180,E1 -1514.021,E2 -1514.021} C_VEL
LIN {X 0,Y 587.153,Z 223.054,A -85,B 0,C 180,E1 -1516.855,E2 -1516.855} C_VEL
LIN {X 0,Y 587.145,Z 225.576,A -85,B 0,C 180,E1 -1517.821,E2 -1517.821} C_VEL
LIN {X 0,Y 587.73,Z 230.397,A -85,B 0,C 180,E1 -1517.921,E2 -1517.921} C_VEL
LIN {X 0,Y 587.68,Z 242.513,A -85,B 0,C 180,E1 -1518.226,E2 -1518.226} C_VEL
LIN {X 0,Y 587.56,Z 254.456,A -85,B 0,C 180,E1 -1518.659,E2 -1518.659} C_VEL
LIN {X 0,Y 587.495,Z 266.207,A -85,B 0,C 180,E1 -1519.227,E2 -1519.227} C_VEL
LIN {X 0,Y 587.445,Z 277.48,A -85,B 0,C 180,E1 -1519.923,E2 -1519.923} C_VEL
LIN {X 0,Y 587.384,Z 287.646,A -85,B 0,C 180,E1 -1520.705,E2 -1520.705} C_VEL
LIN {X 0,Y 587.34,Z 296.776,A -85,B 0,C 180,E1 -1521.571,E2 -1521.571} C_VEL
LIN {X 0,Y 587.259,Z 305.681,A -85,B 0,C 180,E1 -1522.609,E2 -1522.609} C_VEL
LIN {X 0,Y 587.195,Z 312.746,A -85,B 0,C 180,E1 -1523.627,E2 -1523.627} C_VEL
LIN {X 0,Y 587.211,Z 317.681,A -85,B 0,C 180,E1 -1524.506,E2 -1524.506} C_VEL
LIN {X 0,Y 587.188,Z 322.374,A -85,B 0,C 180,E1 -1525.538,E2 -1525.538} C_VEL
LIN {X 0,Y 587.193,Z 325.96,A -85,B 0,C 180,E1 -1526.569,E2 -1526.569} C_VEL
LIN {X 0,Y 587.132,Z 327.803,A -85,B 0,C 180,E1 -1527.256,E2 -1527.256} C_VEL
LIN {X 0,Y 587.141,Z 329.197,A -85,B 0,C 180,E1 -1527.942,E2 -1527.942} C_VEL
LIN {X 0,Y 587.147,Z 330.186,A -85,B 0,C 180,E1 -1528.628,E2 -1528.628} C_VEL
LIN {X 0,Y 587.137,Z 330.987,A -85,B 0,C 180,E1 -1530,E2 -1530} C_VEL
LIN {X 0,Y 587.147,Z 330.186,A -85,B 0,C 180,E1 -1531.372,E2 -1531.372} C_VEL
LIN {X 0,Y 587.141,Z 329.197,A -85,B 0,C 180,E1 -1532.058,E2 -1532.058} C_VEL
LIN {X 0,Y 587.132,Z 327.803,A -85,B 0,C 180,E1 -1532.744,E2 -1532.744} C_VEL
LIN {X 0,Y 587.213,Z 324.892,A -85,B 0,C 180,E1 -1533.774,E2 -1533.774} C_VEL
LIN {X 0,Y 587.147,Z 320.947,A -85,B 0,C 180,E1 -1534.806,E2 -1534.806} C_VEL
LIN {X 0,Y 587.229,Z 315.853,A -85,B 0,C 180,E1 -1535.839,E2 -1535.839} C_VEL
LIN {X 0,Y 587.23,Z 309.469,A -85,B 0,C 180,E1 -1536.874,E2 -1536.874} C_VEL
LIN {X 0,Y 587.287,Z 301.484,A -85,B 0,C 180,E1 -1537.91,E2 -1537.91} C_VEL
LIN {X 0,Y 587.336,Z 293.343,A -85,B 0,C 180,E1 -1538.775,E2 -1538.775} C_VEL
LIN {X 0,Y 587.389,Z 283.383,A -85,B 0,C 180,E1 -1539.643,E2 -1539.643} C_VEL
LIN {X 0,Y 587.428,Z 273.57,A -85,B 0,C 180,E1 -1540.338,E2 -1540.338} C_VEL
LIN {X 0,Y 587.492,Z 262.932,A -85,B 0,C 180,E1 -1540.947,E2 -1540.947} C_VEL
LIN {X 0,Y 587.57,Z 250.644,A -85,B 0,C 180,E1 -1541.494,E2 -1541.494} C_VEL
LIN {X 0,Y 587.682,Z 237.917,A -85,B 0,C 180,E1 -1541.905,E2 -1541.905} C_VEL
LIN {X 0,Y 587.558,Z 228.114,A -85,B 0,C 180,E1 -1542.126,E2 -1542.126} C_VEL
LIN {X 0,Y 587.14,Z 225.468,A -85,B 0,C 180,E1 -1542.201,E2 -1542.201} C_VEL
LIN {X 0,Y 587.17,Z 219.461,A -85,B 0,C 180,E1 -1544.557,E2 -1544.557} C_VEL
LIN {X 0,Y 587.209,Z 212.275,A -85,B 0,C 180,E1 -1547.41,E2 -1547.41} C_VEL
LIN {X 0,Y 587.213,Z 206.885,A -85,B 0,C 180,E1 -1549.579,E2 -1549.579} C_VEL
LIN {X 0,Y 587.268,Z 199.699,A -85,B 0,C 180,E1 -1552.516,E2 -1552.516} C_VEL
LIN {X 0,Y 587.262,Z 192.513,A -85,B 0,C 180,E1 -1555.52,E2 -1555.52} C_VEL
LIN {X 0,Y 587.294,Z 187.123,A -85,B 0,C 180,E1 -1557.82,E2 -1557.82} C_VEL
LIN {X 0,Y 587.345,Z 180.961,A -85,B 0,C 180,E1 -1560.511,E2 -1560.511} C_VEL
LIN {X 0,Y 587.36,Z 174.548,A -85,B 0,C 180,E1 -1563.394,E2 -1563.394} C_VEL
LIN {X 0,Y 587.413,Z 169.158,A -85,B 0,C 180,E1 -1565.891,E2 -1565.891} C_VEL
LIN {X 0,Y 587.475,Z 162.868,A -85,B 0,C 180,E1 -1568.958,E2 -1568.958} C_VEL
LIN {X 0,Y 587.532,Z 158.9,A -85,B 0,C 180,E1 -1571.139,E2 -1571.139} C_VEL
LIN {X 0,Y 587.393,Z 157.304,A -85,B 0,C 180,E1 -1572.114,E2 -1572.114} C_VEL
LIN {X 0,Y 587.304,Z 156.832,A -85,B 0,C 180,E1 -1573.117,E2 -1573.117} C_VEL
LIN {X 0,Y 587.309,Z 156.823,A -85,B 0,C 180,E1 -1576.048,E2 -1576.048} C_VEL
LIN {X 0,Y 587.332,Z 156.829,A -85,B 0,C 180,E1 -1578.924,E2 -1578.924} C_VEL
LIN {X 0,Y 587.32,Z 156.822,A -85,B 0,C 180,E1 -1581.52,E2 -1581.52} C_VEL
LIN {X 0,Y 587.286,Z 156.826,A -85,B 0,C 180,E1 -1584.099,E2 -1584.099} C_VEL
LIN {X 0,Y 587.33,Z 156.828,A -85,B 0,C 180,E1 -1586.603,E2 -1586.603} C_VEL
LIN {X 0,Y 587.333,Z 156.819,A -85,B 0,C 180,E1 -1589.489,E2 -1589.489} C_VEL
LIN {X 0,Y 587.346,Z 156.824,A -85,B 0,C 180,E1 -1592.307,E2 -1592.307} C_VEL
LIN {X 0,Y 587.349,Z 156.817,A -85,B 0,C 180,E1 -1595.419,E2 -1595.419} C_VEL
LIN {X 0,Y 587.317,Z 156.829,A -85,B 0,C 180,E1 -1598.225,E2 -1598.225} C_VEL
LIN {X 0,Y 587.341,Z 156.818,A -85,B 0,C 180,E1 -1601.151,E2 -1601.151} C_VEL
LIN {X 0,Y 587.32,Z 156.828,A -85,B 0,C 180,E1 -1604.024,E2 -1604.024} C_VEL
LIN {X 0,Y 587.351,Z 156.826,A -85,B 0,C 180,E1 -1606.154,E2 -1606.154} C_VEL
LIN {X 0,Y 587.338,Z 156.818,A -85,B 0,C 180,E1 -1608.962,E2 -1608.962} C_VEL
LIN {X 0,Y 587.366,Z 156.821,A -85,B 0,C 180,E1 -1611.744,E2 -1611.744} C_VEL
LIN {X 0,Y 587.344,Z 156.818,A -85,B 0,C 180,E1 -1614.507,E2 -1614.507} C_VEL
LIN {X 0,Y 587.372,Z 156.816,A -85,B 0,C 180,E1 -1617.256,E2 -1617.256} C_VEL
LIN {X 0,Y 587.372,Z 156.819,A -85,B 0,C 180,E1 -1620,E2 -1620} C_VEL
LIN {X 0,Y 587.366,Z 156.815,A -85,B 0,C 180,E1 -1622.743,E2 -1622.743} C_VEL
LIN {X 0,Y 587.353,Z 156.826,A -85,B 0,C 180,E1 -1625.493,E2 -1625.493} C_VEL
LIN {X 0,Y 587.361,Z 156.815,A -85,B 0,C 180,E1 -1628.255,E2 -1628.255} C_VEL
LIN {X 0,Y 587.34,Z 156.824,A -85,B 0,C 180,E1 -1631.133,E2 -1631.133} C_VEL
LIN {X 0,Y 587.357,Z 156.816,A -85,B 0,C 180,E1 -1634.26,E2 -1634.26} C_VEL
LIN {X 0,Y 587.345,Z 156.823,A -85,B 0,C 180,E1 -1637.406,E2 -1637.406} C_VEL
LIN {X 0,Y 587.306,Z 156.822,A -85,B 0,C 180,E1 -1638.311,E2 -1638.311} C_VEL
LIN {X 0,Y 586.664,Z 156.909,A -85,B 0,C 180,E1 -1638.883,E2 -1638.883} C_VEL
LIN {X 0,Y 583.841,Z 157.264,A -85,B 0,C 180,E1 -1639.812,E2 -1639.812} C_VEL
LIN {X 0,Y 581.431,Z 157.566,A -85,B 0,C 180,E1 -1640.559,E2 -1640.559} C_VEL
LIN {X 0,Y 580.376,Z 157.694,A -85,B 0,C 180,E1 -1641.135,E2 -1641.135} C_VEL
LIN {X 0,Y 580.28,Z 157.702,A -85,B 0,C 180,E1 -1641.331,E2 -1641.331} C_VEL
LIN {X 0,Y 580.294,Z 157.697,A -85,B 0,C 180,E1 -1644.316,E2 -1644.316} C_VEL
LIN {X 0,Y 580.27,Z 157.704,A -85,B 0,C 180,E1 -1646.623,E2 -1646.623} C_VEL
LIN {X 0,Y 580.299,Z 157.697,A -85,B 0,C 180,E1 -1649.311,E2 -1649.311} C_VEL
LIN {X 0,Y 580.294,Z 157.698,A -85,B 0,C 180,E1 -1652.2,E2 -1652.2} C_VEL
LIN {X 0,Y 580.295,Z 157.705,A -85,B 0,C 180,E1 -1654.695,E2 -1654.695} C_VEL
LIN {X 0,Y 580.293,Z 157.697,A -85,B 0,C 180,E1 -1657.268,E2 -1657.268} C_VEL
LIN {X 0,Y 580.299,Z 157.701,A -85,B 0,C 180,E1 -1660.272,E2 -1660.272} C_VEL
LIN {X 0,Y 580.275,Z 157.703,A -85,B 0,C 180,E1 -1662.706,E2 -1662.706} C_VEL
LIN {X 0,Y 580.263,Z 157.7,A -85,B 0,C 180,E1 -1665.609,E2 -1665.609} C_VEL
LIN {X 0,Y 580.308,Z 157.704,A -85,B 0,C 180,E1 -1668.234,E2 -1668.234} C_VEL
LIN {X 0,Y 580.284,Z 157.697,A -85,B 0,C 180,E1 -1670.966,E2 -1670.966} C_VEL
LIN {X 0,Y 580.292,Z 157.698,A -85,B 0,C 180,E1 -1673.599,E2 -1673.599} C_VEL
LIN {X 0,Y 580.315,Z 157.701,A -85,B 0,C 180,E1 -1676.146,E2 -1676.146} C_VEL
LIN {X 0,Y 580.285,Z 157.698,A -85,B 0,C 180,E1 -1678.616,E2 -1678.616} C_VEL
LIN {X 0,Y 580.29,Z 157.696,A -85,B 0,C 180,E1 -1681.024,E2 -1681.024} C_VEL
LIN {X 0,Y 580.287,Z 157.704,A -85,B 0,C 180,E1 -1683.666,E2 -1683.666} C_VEL
LIN {X 0,Y 580.297,Z 157.705,A -85,B 0,C 180,E1 -1685.684,E2 -1685.684} C_VEL
LIN {X 0,Y 580.271,Z 157.704,A -85,B 0,C 180,E1 -1687.948,E2 -1687.948} C_VEL
LIN {X 0,Y 580.315,Z 157.694,A -85,B 0,C 180,E1 -1690.914,E2 -1690.914} C_VEL
LIN {X 0,Y 580.277,Z 157.703,A -85,B 0,C 180,E1 -1693.826,E2 -1693.826} C_VEL
LIN {X 0,Y 580.322,Z 157.695,A -85,B 0,C 180,E1 -1695.983,E2 -1695.983} C_VEL
LIN {X 0,Y 580.301,Z 157.698,A -85,B 0,C 180,E1 -1698.827,E2 -1698.827} C_VEL
LIN {X 0,Y 580.331,Z 157.695,A -85,B 0,C 180,E1 -1701.644,E2 -1701.644} C_VEL
LIN {X 0,Y 580.328,Z 157.693,A -85,B 0,C 180,E1 -1704.44,E2 -1704.44} C_VEL
LIN {X 0,Y 580.343,Z 157.69,A -85,B 0,C 180,E1 -1707.918,E2 -1707.918} C_VEL
LIN {X 0,Y 580.359,Z 157.694,A -85,B 0,C 180,E1 -1710.694,E2 -1710.694} C_VEL
LIN {X 0,Y 580.281,Z 157.7,A -85,B 0,C 180,E1 -1713.472,E2 -1713.472} C_VEL
LIN {X 0,Y 580.328,Z 157.693,A -85,B 0,C 180,E1 -1715.56,E2 -1715.56} C_VEL
LIN {X 0,Y 580.331,Z 157.695,A -85,B 0,C 180,E1 -1718.356,E2 -1718.356} C_VEL
LIN {X 0,Y 580.296,Z 157.698,A -85,B 0,C 180,E1 -1721.191,E2 -1721.191} C_VEL
LIN {X 0,Y 580.322,Z 157.695,A -85,B 0,C 180,E1 -1724.017,E2 -1724.017} C_VEL
LIN {X 0,Y 580.308,Z 157.698,A -85,B 0,C 180,E1 -1726.914,E2 -1726.914} C_VEL
LIN {X 0,Y 580.303,Z 157.696,A -85,B 0,C 180,E1 -1729.822,E2 -1729.822} C_VEL
LIN {X 0,Y 580.291,Z 157.699,A -85,B 0,C 180,E1 -1732.802,E2 -1732.802} C_VEL
LIN {X 0,Y 580.302,Z 157.695,A -85,B 0,C 180,E1 -1735.08,E2 -1735.08} C_VEL
LIN {X 0,Y 580.297,Z 157.705,A -85,B 0,C 180,E1 -1738.185,E2 -1738.185} C_VEL
LIN {X 0,Y 580.295,Z 157.697,A -85,B 0,C 180,E1 -1740.697,E2 -1740.697} C_VEL
LIN {X 0,Y 580.299,Z 157.696,A -85,B 0,C 180,E1 -1743.316,E2 -1743.316} C_VEL
LIN {X 0,Y 580.322,Z 157.699,A -85,B 0,C 180,E1 -1745.767,E2 -1745.767} C_VEL
LIN {X 0,Y 580.284,Z 157.702,A -85,B 0,C 180,E1 -1748.146,E2 -1748.146} C_VEL
LIN {X 0,Y 580.298,Z 157.695,A -85,B 0,C 180,E1 -1750.843,E2 -1750.843} C_VEL
LIN {X 0,Y 580.272,Z 157.708,A -85,B 0,C 180,E1 -1753.658,E2 -1753.658} C_VEL
LIN {X 0,Y 580.279,Z 157.697,A -85,B 0,C 180,E1 -1756.608,E2 -1756.608} C_VEL
LIN {X 0,Y 580.294,Z 157.7,A -85,B 0,C 180,E1 -1759.157,E2 -1759.157} C_VEL
LIN {X 0,Y 580.284,Z 157.7,A -85,B 0,C 180,E1 -1761.927,E2 -1761.927} C_VEL
LIN {X 0,Y 580.3,Z 157.695,A -85,B 0,C 180,E1 -1764.457,E2 -1764.457} C_VEL
LIN {X 0,Y 580.285,Z 157.701,A -85,B 0,C 180,E1 -1766.975,E2 -1766.975} C_VEL
LIN {X 0,Y 580.3,Z 157.701,A -85,B 0,C 180,E1 -1769.426,E2 -1769.426} C_VEL
LIN {X 0,Y 580.313,Z 157.693,A -85,B 0,C 180,E1 -1772.137,E2 -1772.137} C_VEL
LIN {X 0,Y 580.314,Z 157.699,A -85,B 0,C 180,E1 -1775.27,E2 -1775.27} C_VEL
LIN {X 0,Y 580.266,Z 157.699,A -85,B 0,C 180,E1 -1777.948,E2 -1777.948} C_VEL
LIN {X 0,Y 580.311,Z 157.703,A -85,B 0,C 180,E1 -1780.914,E2 -1780.914} C_VEL
LIN {X 0,Y 580.275,Z 157.698,A -85,B 0,C 180,E1 -1783.826,E2 -1783.826} C_VEL
LIN {X 0,Y 580.319,Z 157.693,A -85,B 0,C 180,E1 -1785.983,E2 -1785.983} C_VEL
LIN {X 0,Y 580.297,Z 157.702,A -85,B 0,C 180,E1 -1788.827,E2 -1788.827} C_VEL
LIN {X 0,Y 580.326,Z 157.692,A -85,B 0,C 180,E1 -1791.644,E2 -1791.644} C_VEL
LIN {X 0,Y 580.318,Z 157.702,A -85,B 0,C 180,E1 -1794.441,E2 -1794.441} C_VEL
LIN {X 0,Y 580.332,Z 157.691,A -85,B 0,C 180,E1 -1797.224,E2 -1797.224} C_VEL
LIN {X 0,Y 580.341,Z 157.694,A -85,B 0,C 180,E1 -1800,E2 -1800} C_VEL
LIN {X 0,Y 580.338,Z 157.692,A -85,B 0,C 180,E1 -1802.777,E2 -1802.777} C_VEL
LIN {X 0,Y 580.311,Z 157.695,A -85,B 0,C 180,E1 -1805.56,E2 -1805.56} C_VEL
LIN {X 0,Y 580.329,Z 157.696,A -85,B 0,C 180,E1 -1808.356,E2 -1808.356} C_VEL
LIN {X 0,Y 580.294,Z 157.696,A -85,B 0,C 180,E1 -1811.192,E2 -1811.192} C_VEL
LIN {X 0,Y 580.319,Z 157.7,A -85,B 0,C 180,E1 -1814.017,E2 -1814.017} C_VEL
LIN {X 0,Y 580.307,Z 157.694,A -85,B 0,C 180,E1 -1816.914,E2 -1816.914} C_VEL
LIN {X 0,Y 580.298,Z 157.703,A -85,B 0,C 180,E1 -1819.823,E2 -1819.823} C_VEL
LIN {X 0,Y 580.289,Z 157.696,A -85,B 0,C 180,E1 -1822.803,E2 -1822.803} C_VEL
LIN {X 0,Y 580.303,Z 157.697,A -85,B 0,C 180,E1 -1825.08,E2 -1825.08} C_VEL
LIN {X 0,Y 580.29,Z 157.697,A -85,B 0,C 180,E1 -1828.186,E2 -1828.186} C_VEL
LIN {X 0,Y 580.282,Z 157.698,A -85,B 0,C 180,E1 -1830.696,E2 -1830.696} C_VEL
LIN {X 0,Y 580.299,Z 157.705,A -85,B 0,C 180,E1 -1833.317,E2 -1833.317} C_VEL
LIN {X 0,Y 580.241,Z 157.705,A -85,B 0,C 180,E1 -1835.757,E2 -1835.757} C_VEL
LIN {X 0,Y 580.282,Z 157.698,A -85,B 0,C 180,E1 -1838.147,E2 -1838.147} C_VEL
LIN {X 0,Y 580.295,Z 157.702,A -85,B 0,C 180,E1 -1840.844,E2 -1840.844} C_VEL
LIN {X 0,Y 580.267,Z 157.702,A -85,B 0,C 180,E1 -1843.659,E2 -1843.659} C_VEL
LIN {X 0,Y 580.243,Z 157.711,A -85,B 0,C 180,E1 -1846.613,E2 -1846.613} C_VEL
LIN {X 0,Y 580.257,Z 157.709,A -85,B 0,C 180,E1 -1847.293,E2 -1847.293} C_VEL
LIN {X 0,Y 580.56,Z 160.789,A -85,B 0,C 180,E1 -1849.18,E2 -1849.18} C_VEL
LIN {X 0,Y 580.438,Z 165.757,A -85,B 0,C 180,E1 -1851.909,E2 -1851.909} C_VEL
LIN {X 0,Y 580.393,Z 170.955,A -85,B 0,C 180,E1 -1854.463,E2 -1854.463} C_VEL
LIN {X 0,Y 580.348,Z 176.344,A -85,B 0,C 180,E1 -1856.979,E2 -1856.979} C_VEL
LIN {X 0,Y 580.305,Z 181.734,A -85,B 0,C 180,E1 -1859.426,E2 -1859.426} C_VEL
LIN {X 0,Y 580.245,Z 187.9,A -85,B 0,C 180,E1 -1862.152,E2 -1862.152} C_VEL
LIN {X 0,Y 580.228,Z 194.309,A -85,B 0,C 180,E1 -1864.917,E2 -1864.917} C_VEL
LIN {X 0,Y 580.198,Z 201.495,A -85,B 0,C 180,E1 -1867.945,E2 -1867.945} C_VEL
LIN {X 0,Y 580.182,Z 208.682,A -85,B 0,C 180,E1 -1870.91,E2 -1870.91} C_VEL
LIN {X 0,Y 580.107,Z 215.868,A -85,B 0,C 180,E1 -1873.821,E2 -1873.821} C_VEL
LIN {X 0,Y 580.066,Z 223.054,A -85,B 0,C 180,E1 -1876.691,E2 -1876.691} C_VEL
LIN {X 0,Y 580.07,Z 225.55,A -85,B 0,C 180,E1 -1877.67,E2 -1877.67} C_VEL
LIN {X 0,Y 580.785,Z 231.534,A -85,B 0,C 180,E1 -1877.797,E2 -1877.797} C_VEL
LIN {X 0,Y 580.703,Z 243.847,A -85,B 0,C 180,E1 -1878.127,E2 -1878.127} C_VEL
LIN {X 0,Y 580.573,Z 256.193,A -85,B 0,C 180,E1 -1878.598,E2 -1878.598} C_VEL
LIN {X 0,Y 580.499,Z 267.773,A -85,B 0,C 180,E1 -1879.184,E2 -1879.184} C_VEL
LIN {X 0,Y 580.438,Z 278.75,A -85,B 0,C 180,E1 -1879.888,E2 -1879.888} C_VEL
LIN {X 0,Y 580.333,Z 289.588,A -85,B 0,C 180,E1 -1880.766,E2 -1880.766} C_VEL
LIN {X 0,Y 580.263,Z 298.398,A -85,B 0,C 180,E1 -1881.643,E2 -1881.643} C_VEL
LIN {X 0,Y 580.175,Z 307.005,A -85,B 0,C 180,E1 -1882.693,E2 -1882.693} C_VEL
LIN {X 0,Y 580.135,Z 313.87,A -85,B 0,C 180,E1 -1883.741,E2 -1883.741} C_VEL
LIN {X 0,Y 580.086,Z 319.364,A -85,B 0,C 180,E1 -1884.787,E2 -1884.787} C_VEL
LIN {X 0,Y 580.105,Z 323.669,A -85,B 0,C 180,E1 -1885.832,E2 -1885.832} C_VEL
LIN {X 0,Y 580.123,Z 325.962,A -85,B 0,C 180,E1 -1886.527,E2 -1886.527} C_VEL
LIN {X 0,Y 580.043,Z 327.8,A -85,B 0,C 180,E1 -1887.222,E2 -1887.222} C_VEL
LIN {X 0,Y 580.047,Z 330.187,A -85,B 0,C 180,E1 -1888.611,E2 -1888.611} C_VEL
LIN {X 0,Y 580.04,Z 330.782,A -85,B 0,C 180,E1 -1889.306,E2 -1889.306} C_VEL
LIN {X 0,Y 580.037,Z 330.983,A -85,B 0,C 180,E1 -1890,E2 -1890} C_VEL
LIN {X 0,Y 580.04,Z 330.782,A -85,B 0,C 180,E1 -1890.694,E2 -1890.694} C_VEL
LIN {X 0,Y 580.047,Z 330.187,A -85,B 0,C 180,E1 -1891.389,E2 -1891.389} C_VEL
LIN {X 0,Y 580.043,Z 327.8,A -85,B 0,C 180,E1 -1892.778,E2 -1892.778} C_VEL
LIN {X 0,Y 580.11,Z 324.89,A -85,B 0,C 180,E1 -1893.821,E2 -1893.821} C_VEL
LIN {X 0,Y 580.053,Z 320.943,A -85,B 0,C 180,E1 -1894.865,E2 -1894.865} C_VEL
LIN {X 0,Y 580.161,Z 315.849,A -85,B 0,C 180,E1 -1895.91,E2 -1895.91} C_VEL
LIN {X 0,Y 580.157,Z 309.465,A -85,B 0,C 180,E1 -1896.958,E2 -1896.958} C_VEL
LIN {X 0,Y 580.242,Z 301.486,A -85,B 0,C 180,E1 -1898.007,E2 -1898.007} C_VEL
LIN {X 0,Y 580.305,Z 293.345,A -85,B 0,C 180,E1 -1898.883,E2 -1898.883} C_VEL
LIN {X 0,Y 580.357,Z 283.377,A -85,B 0,C 180,E1 -1899.761,E2 -1899.761} C_VEL
LIN {X 0,Y 580.44,Z 273.562,A -85,B 0,C 180,E1 -1900.464,E2 -1900.464} C_VEL
LIN {X 0,Y 580.522,Z 262.934,A -85,B 0,C 180,E1 -1901.08,E2 -1901.08} C_VEL
LIN {X 0,Y 580.638,Z 250.142,A -85,B 0,C 180,E1 -1901.653,E2 -1901.653} C_VEL
LIN {X 0,Y 580.736,Z 237.902,A -85,B 0,C 180,E1 -1902.049,E2 -1902.049} C_VEL
LIN {X 0,Y 580.665,Z 229.116,A -85,B 0,C 180,E1 -1902.253,E2 -1902.253} C_VEL
LIN {X 0,Y 580.074,Z 225.468,A -85,B 0,C 180,E1 -1902.352,E2 -1902.352} C_VEL
LIN {X 0,Y 580.099,Z 219.461,A -85,B 0,C 180,E1 -1904.739,E2 -1904.739} C_VEL
LIN {X 0,Y 580.139,Z 212.275,A -85,B 0,C 180,E1 -1907.629,E2 -1907.629} C_VEL
LIN {X 0,Y 580.157,Z 206.885,A -85,B 0,C 180,E1 -1909.827,E2 -1909.827} C_VEL
LIN {X 0,Y 580.198,Z 201.495,A -85,B 0,C 180,E1 -1912.055,E2 -1912.055} C_VEL
LIN {X 0,Y 580.228,Z 194.309,A -85,B 0,C 180,E1 -1915.083,E2 -1915.083} C_VEL
LIN {X 0,Y 580.245,Z 187.9,A -85,B 0,C 180,E1 -1917.848,E2 -1917.848} C_VEL
LIN {X 0,Y 580.298,Z 181.463,A -85,B 0,C 180,E1 -1920.696,E2 -1920.696} C_VEL
LIN {X 0,Y 580.356,Z 175.687,A -85,B 0,C 180,E1 -1923.324,E2 -1923.324} C_VEL
LIN {X 0,Y 580.386,Z 169.158,A -85,B 0,C 180,E1 -1926.394,E2 -1926.394} C_VEL
LIN {X 0,Y 580.489,Z 163.693,A -85,B 0,C 180,E1 -1929.208,E2 -1929.208} C_VEL
LIN {X 0,Y 580.524,Z 159.88,A -85,B 0,C 180,E1 -1931.358,E2 -1931.358} C_VEL
LIN {X 0,Y 580.257,Z 157.709,A -85,B 0,C 180,E1 -1932.707,E2 -1932.707} C_VEL
LIN {X 0,Y 580.256,Z 157.704,A -85,B 0,C 180,E1 -1935.61,E2 -1935.61} C_VEL
LIN {X 0,Y 580.27,Z 157.701,A -85,B 0,C 180,E1 -1938.23,E2 -1938.23} C_VEL
LIN {X 0,Y 580.281,Z 157.706,A -85,B 0,C 180,E1 -1940.965,E2 -1940.965} C_VEL
LIN {X 0,Y 580.263,Z 157.7,A -85,B 0,C 180,E1 -1943.596,E2 -1943.596} C_VEL
LIN {X 0,Y 580.31,Z 157.696,A -85,B 0,C 180,E1 -1946.144,E2 -1946.144} C_VEL
LIN {X 0,Y 580.275,Z 157.708,A -85,B 0,C 180,E1 -1948.614,E2 -1948.614} C_VEL
LIN {X 0,Y 580.283,Z 157.7,A -85,B 0,C 180,E1 -1951.023,E2 -1951.023} C_VEL
LIN {X 0,Y 580.281,Z 157.697,A -85,B 0,C 180,E1 -1953.666,E2 -1953.666} C_VEL
LIN {X 0,Y 580.297,Z 157.696,A -85,B 0,C 180,E1 -1955.683,E2 -1955.683} C_VEL
LIN {X 0,Y 580.267,Z 157.703,A -85,B 0,C 180,E1 -1957.947,E2 -1957.947} C_VEL
LIN {X 0,Y 580.294,Z 157.697,A -85,B 0,C 180,E1 -1960.913,E2 -1960.913} C_VEL
LIN {X 0,Y 580.275,Z 157.702,A -85,B 0,C 180,E1 -1963.825,E2 -1963.825} C_VEL
LIN {X 0,Y 580.319,Z 157.7,A -85,B 0,C 180,E1 -1965.983,E2 -1965.983} C_VEL
LIN {X 0,Y 580.299,Z 157.695,A -85,B 0,C 180,E1 -1968.826,E2 -1968.826} C_VEL
LIN {X 0,Y 580.329,Z 157.696,A -85,B 0,C 180,E1 -1971.644,E2 -1971.644} C_VEL
LIN {X 0,Y 580.311,Z 157.695,A -85,B 0,C 180,E1 -1974.44,E2 -1974.44} C_VEL
LIN {X 0,Y 580.337,Z 157.692,A -85,B 0,C 180,E1 -1977.223,E2 -1977.223} C_VEL
LIN {X 0,Y 580.341,Z 157.694,A -85,B 0,C 180,E1 -1980,E2 -1980} C_VEL
LIN {X 0,Y 580.332,Z 157.691,A -85,B 0,C 180,E1 -1982.776,E2 -1982.776} C_VEL
LIN {X 0,Y 580.318,Z 157.702,A -85,B 0,C 180,E1 -1985.559,E2 -1985.559} C_VEL
LIN {X 0,Y 580.326,Z 157.692,A -85,B 0,C 180,E1 -1988.356,E2 -1988.356} C_VEL
LIN {X 0,Y 580.292,Z 157.703,A -85,B 0,C 180,E1 -1991.191,E2 -1991.191} C_VEL
LIN {X 0,Y 580.319,Z 157.693,A -85,B 0,C 180,E1 -1994.017,E2 -1994.017} C_VEL
LIN {X 0,Y 580.306,Z 157.7,A -85,B 0,C 180,E1 -1996.914,E2 -1996.914} C_VEL
LIN {X 0,Y 580.3,Z 157.695,A -85,B 0,C 180,E1 -1999.822,E2 -1999.822} C_VEL
LIN {X 0,Y 580.28,Z 157.702,A -85,B 0,C 180,E1 -2001.331,E2 -2001.331} C_VEL
LIN {X 0,Y 579.581,Z 157.787,A -85,B 0,C 180,E1 -2001.91,E2 -2001.91} C_VEL
LIN {X 0,Y 576.703,Z 158.15,A -85,B 0,C 180,E1 -2002.85,E2 -2002.85} C_VEL
LIN {X 0,Y 574.309,Z 158.444,A -85,B 0,C 180,E1 -2003.606,E2 -2003.606} C_VEL
LIN {X 0,Y 573.31,Z 158.566,A -85,B 0,C 180,E1 -2004.19,E2 -2004.19} C_VEL
LIN {X 0,Y 573.243,Z 158.576,A -85,B 0,C 180,E1 -2004.387,E2 -2004.387} C_VEL
LIN {X 0,Y 573.244,Z 158.582,A -85,B 0,C 180,E1 -2006.976,E2 -2006.976} C_VEL
LIN {X 0,Y 573.245,Z 158.575,A -85,B 0,C 180,E1 -2009.489,E2 -2009.489} C_VEL
LIN {X 0,Y 573.247,Z 158.576,A -85,B 0,C 180,E1 -2012.229,E2 -2012.229} C_VEL
LIN {X 0,Y 573.245,Z 158.581,A -85,B 0,C 180,E1 -2014.774,E2 -2014.774} C_VEL
LIN {X 0,Y 573.247,Z 158.575,A -85,B 0,C 180,E1 -2017.166,E2 -2017.166} C_VEL
LIN {X 0,Y 573.243,Z 158.574,A -85,B 0,C 180,E1 -2019.607,E2 -2019.607} C_VEL
LIN {X 0,Y 573.237,Z 158.581,A -85,B 0,C 180,E1 -2022.642,E2 -2022.642} C_VEL
LIN {X 0,Y 573.228,Z 158.577,A -85,B 0,C 180,E1 -2025.667,E2 -2025.667} C_VEL
LIN {X 0,Y 573.238,Z 158.579,A -85,B 0,C 180,E1 -2028.544,E2 -2028.544} C_VEL
LIN {X 0,Y 573.243,Z 158.574,A -85,B 0,C 180,E1 -2031.299,E2 -2031.299} C_VEL
LIN {X 0,Y 573.26,Z 158.581,A -85,B 0,C 180,E1 -2034.011,E2 -2034.011} C_VEL
LIN {X 0,Y 573.28,Z 158.572,A -85,B 0,C 180,E1 -2036.519,E2 -2036.519} C_VEL
LIN {X 0,Y 573.239,Z 158.575,A -85,B 0,C 180,E1 -2039.115,E2 -2039.115} C_VEL
LIN {X 0,Y 573.26,Z 158.579,A -85,B 0,C 180,E1 -2041.969,E2 -2041.969} C_VEL
LIN {X 0,Y 573.249,Z 158.573,A -85,B 0,C 180,E1 -2044.59,E2 -2044.59} C_VEL
LIN {X 0,Y 573.234,Z 158.585,A -85,B 0,C 180,E1 -2047.662,E2 -2047.662} C_VEL
LIN {X 0,Y 573.274,Z 158.57,A -85,B 0,C 180,E1 -2050.728,E2 -2050.728} C_VEL
LIN {X 0,Y 573.249,Z 158.582,A -85,B 0,C 180,E1 -2053.622,E2 -2053.622} C_VEL
LIN {X 0,Y 573.27,Z 158.575,A -85,B 0,C 180,E1 -2055.807,E2 -2055.807} C_VEL
LIN {X 0,Y 573.259,Z 158.574,A -85,B 0,C 180,E1 -2058.745,E2 -2058.745} C_VEL
LIN {X 0,Y 573.287,Z 158.575,A -85,B 0,C 180,E1 -2061.541,E2 -2061.541} C_VEL
LIN {X 0,Y 573.296,Z 158.568,A -85,B 0,C 180,E1 -2064.372,E2 -2064.372} C_VEL
LIN {X 0,Y 573.313,Z 158.566,A -85,B 0,C 180,E1 -2067.892,E2 -2067.892} C_VEL
LIN {X 0,Y 573.33,Z 158.57,A -85,B 0,C 180,E1 -2070.702,E2 -2070.702} C_VEL
LIN {X 0,Y 573.303,Z 158.575,A -85,B 0,C 180,E1 -2072.811,E2 -2072.811} C_VEL
LIN {X 0,Y 573.296,Z 158.568,A -85,B 0,C 180,E1 -2075.628,E2 -2075.628} C_VEL
LIN {X 0,Y 573.287,Z 158.575,A -85,B 0,C 180,E1 -2078.459,E2 -2078.459} C_VEL
LIN {X 0,Y 573.268,Z 158.573,A -85,B 0,C 180,E1 -2081.312,E2 -2081.312} C_VEL
LIN {X 0,Y 573.269,Z 158.575,A -85,B 0,C 180,E1 -2084.193,E2 -2084.193} C_VEL
LIN {X 0,Y 573.255,Z 158.575,A -85,B 0,C 180,E1 -2087.111,E2 -2087.111} C_VEL
LIN {X 0,Y 573.25,Z 158.578,A -85,B 0,C 180,E1 -2090.076,E2 -2090.076} C_VEL
LIN {X 0,Y 573.23,Z 158.576,A -85,B 0,C 180,E1 -2093.099,E2 -2093.099} C_VEL
LIN {X 0,Y 573.249,Z 158.573,A -85,B 0,C 180,E1 -2095.41,E2 -2095.41} C_VEL
LIN {X 0,Y 573.26,Z 158.579,A -85,B 0,C 180,E1 -2098.031,E2 -2098.031} C_VEL
LIN {X 0,Y 573.239,Z 158.575,A -85,B 0,C 180,E1 -2100.885,E2 -2100.885} C_VEL
LIN {X 0,Y 573.257,Z 158.575,A -85,B 0,C 180,E1 -2103.524,E2 -2103.524} C_VEL
LIN {X 0,Y 573.256,Z 158.58,A -85,B 0,C 180,E1 -2106.048,E2 -2106.048} C_VEL
LIN {X 0,Y 573.244,Z 158.574,A -85,B 0,C 180,E1 -2108.701,E2 -2108.701} C_VEL
LIN {X 0,Y 573.248,Z 158.58,A -85,B 0,C 180,E1 -2111.596,E2 -2111.596} C_VEL
LIN {X 0,Y 573.228,Z 158.577,A -85,B 0,C 180,E1 -2114.333,E2 -2114.333} C_VEL
LIN {X 0,Y 573.237,Z 158.581,A -85,B 0,C 180,E1 -2117.358,E2 -2117.358} C_VEL
LIN {X 0,Y 573.242,Z 158.574,A -85,B 0,C 180,E1 -2120.393,E2 -2120.393} C_VEL
LIN {X 0,Y 573.249,Z 158.578,A -85,B 0,C 180,E1 -2123.078,E2 -2123.078} C_VEL
LIN {X 0,Y 573.267,Z 158.575,A -85,B 0,C 180,E1 -2125.672,E2 -2125.672} C_VEL
LIN {X 0,Y 573.239,Z 158.574,A -85,B 0,C 180,E1 -2128.185,E2 -2128.185} C_VEL
LIN {X 0,Y 573.262,Z 158.574,A -85,B 0,C 180,E1 -2130.635,E2 -2130.635} C_VEL
LIN {X 0,Y 573.244,Z 158.582,A -85,B 0,C 180,E1 -2133.024,E2 -2133.024} C_VEL
LIN {X 0,Y 573.268,Z 158.576,A -85,B 0,C 180,E1 -2135.366,E2 -2135.366} C_VEL
LIN {X 0,Y 573.224,Z 158.578,A -85,B 0,C 180,E1 -2138.42,E2 -2138.42} C_VEL
LIN {X 0,Y 573.273,Z 158.577,A -85,B 0,C 180,E1 -2140.728,E2 -2140.728} C_VEL
LIN {X 0,Y 573.251,Z 158.573,A -85,B 0,C 180,E1 -2143.622,E2 -2143.622} C_VEL
LIN {X 0,Y 573.232,Z 158.582,A -85,B 0,C 180,E1 -2146.53,E2 -2146.53} C_VEL
LIN {X 0,Y 573.255,Z 158.581,A -85,B 0,C 180,E1 -2148.745,E2 -2148.745} C_VEL
LIN {X 0,Y 573.282,Z 158.569,A -85,B 0,C 180,E1 -2151.541,E2 -2151.541} C_VEL
LIN {X 0,Y 573.285,Z 158.577,A -85,B 0,C 180,E1 -2154.372,E2 -2154.372} C_VEL
LIN {X 0,Y 573.299,Z 158.567,A -85,B 0,C 180,E1 -2157.19,E2 -2157.19} C_VEL
LIN {X 0,Y 573.311,Z 158.57,A -85,B 0,C 180,E1 -2160,E2 -2160} C_VEL
LIN {X 0,Y 573.303,Z 158.568,A -85,B 0,C 180,E1 -2162.811,E2 -2162.811} C_VEL
LIN {X 0,Y 573.279,Z 158.572,A -85,B 0,C 180,E1 -2165.629,E2 -2165.629} C_VEL
LIN {X 0,Y 573.284,Z 158.572,A -85,B 0,C 180,E1 -2168.46,E2 -2168.46} C_VEL
LIN {X 0,Y 573.266,Z 158.572,A -85,B 0,C 180,E1 -2171.312,E2 -2171.312} C_VEL
LIN {X 0,Y 573.267,Z 158.576,A -85,B 0,C 180,E1 -2174.193,E2 -2174.193} C_VEL
LIN {X 0,Y 573.253,Z 158.574,A -85,B 0,C 180,E1 -2177.112,E2 -2177.112} C_VEL
LIN {X 0,Y 573.246,Z 158.578,A -85,B 0,C 180,E1 -2180.077,E2 -2180.077} C_VEL
LIN {X 0,Y 573.23,Z 158.578,A -85,B 0,C 180,E1 -2183.1,E2 -2183.1} C_VEL
LIN {X 0,Y 573.246,Z 158.581,A -85,B 0,C 180,E1 -2185.411,E2 -2185.411} C_VEL
LIN {X 0,Y 573.228,Z 158.576,A -85,B 0,C 180,E1 -2188.565,E2 -2188.565} C_VEL
LIN {X 0,Y 573.224,Z 158.58,A -85,B 0,C 180,E1 -2190.994,E2 -2190.994} C_VEL
LIN {X 0,Y 573.259,Z 158.579,A -85,B 0,C 180,E1 -2193.525,E2 -2193.525} C_VEL
LIN {X 0,Y 573.21,Z 158.579,A -85,B 0,C 180,E1 -2196.052,E2 -2196.052} C_VEL
LIN {X 0,Y 573.242,Z 158.578,A -85,B 0,C 180,E1 -2198.702,E2 -2198.702} C_VEL
LIN {X 0,Y 573.222,Z 158.58,A -85,B 0,C 180,E1 -2201.593,E2 -2201.593} C_VEL
LIN {X 0,Y 573.222,Z 158.581,A -85,B 0,C 180,E1 -2204.335,E2 -2204.335} C_VEL
LIN {X 0,Y 573.208,Z 158.587,A -85,B 0,C 180,E1 -2206.639,E2 -2206.639} C_VEL
LIN {X 0,Y 573.385,Z 159.538,A -85,B 0,C 180,E1 -2207.614,E2 -2207.614} C_VEL
LIN {X 0,Y 573.574,Z 162.677,A -85,B 0,C 180,E1 -2209.504,E2 -2209.504} C_VEL
LIN {X 0,Y 573.413,Z 167.573,A -85,B 0,C 180,E1 -2212.207,E2 -2212.207} C_VEL
LIN {X 0,Y 573.328,Z 172.751,A -85,B 0,C 180,E1 -2214.821,E2 -2214.821} C_VEL
LIN {X 0,Y 573.288,Z 178.141,A -85,B 0,C 180,E1 -2217.358,E2 -2217.358} C_VEL
LIN {X 0,Y 573.247,Z 183.53,A -85,B 0,C 180,E1 -2219.824,E2 -2219.824} C_VEL
LIN {X 0,Y 573.189,Z 188.92,A -85,B 0,C 180,E1 -2222.23,E2 -2222.23} C_VEL
LIN {X 0,Y 573.173,Z 195.598,A -85,B 0,C 180,E1 -2225.143,E2 -2225.143} C_VEL
LIN {X 0,Y 573.117,Z 201.496,A -85,B 0,C 180,E1 -2227.658,E2 -2227.658} C_VEL
LIN {X 0,Y 573.077,Z 206.885,A -85,B 0,C 180,E1 -2229.917,E2 -2229.917} C_VEL
LIN {X 0,Y 573.052,Z 214.071,A -85,B 0,C 180,E1 -2232.882,E2 -2232.882} C_VEL
LIN {X 0,Y 573.025,Z 221.257,A -85,B 0,C 180,E1 -2235.801,E2 -2235.801} C_VEL
LIN {X 0,Y 572.984,Z 225.524,A -85,B 0,C 180,E1 -2237.515,E2 -2237.515} C_VEL
LIN {X 0,Y 573.843,Z 231.535,A -85,B 0,C 180,E1 -2237.647,E2 -2237.647} C_VEL
LIN {X 0,Y 573.758,Z 243.839,A -85,B 0,C 180,E1 -2237.981,E2 -2237.981} C_VEL
LIN {X 0,Y 573.637,Z 255.362,A -85,B 0,C 180,E1 -2238.422,E2 -2238.422} C_VEL
LIN {X 0,Y 573.507,Z 266.574,A -85,B 0,C 180,E1 -2238.982,E2 -2238.982} C_VEL
LIN {X 0,Y 573.44,Z 278.75,A -85,B 0,C 180,E1 -2239.764,E2 -2239.764} C_VEL
LIN {X 0,Y 573.307,Z 287.644,A -85,B 0,C 180,E1 -2240.474,E2 -2240.474} C_VEL
LIN {X 0,Y 573.214,Z 296.769,A -85,B 0,C 180,E1 -2241.362,E2 -2241.362} C_VEL
LIN {X 0,Y 573.16,Z 304.317,A -85,B 0,C 180,E1 -2242.248,E2 -2242.248} C_VEL
LIN {X 0,Y 573.065,Z 311.701,A -85,B 0,C 180,E1 -2243.304,E2 -2243.304} C_VEL
LIN {X 0,Y 573.068,Z 317.682,A -85,B 0,C 180,E1 -2244.37,E2 -2244.37} C_VEL
LIN {X 0,Y 573.028,Z 322.376,A -85,B 0,C 180,E1 -2245.428,E2 -2245.428} C_VEL
LIN {X 0,Y 573.022,Z 325.963,A -85,B 0,C 180,E1 -2246.484,E2 -2246.484} C_VEL
LIN {X 0,Y 572.959,Z 327.797,A -85,B 0,C 180,E1 -2247.188,E2 -2247.188} C_VEL
LIN {X 0,Y 572.946,Z 330.188,A -85,B 0,C 180,E1 -2248.594,E2 -2248.594} C_VEL
LIN {X 0,Y 572.941,Z 330.782,A -85,B 0,C 180,E1 -2249.297,E2 -2249.297} C_VEL
LIN {X 0,Y 572.938,Z 330.979,A -85,B 0,C 180,E1 -2250,E2 -2250} C_VEL
LIN {X 0,Y 572.941,Z 330.782,A -85,B 0,C 180,E1 -2250.703,E2 -2250.703} C_VEL
LIN {X 0,Y 572.946,Z 330.188,A -85,B 0,C 180,E1 -2251.406,E2 -2251.406} C_VEL
LIN {X 0,Y 572.959,Z 327.797,A -85,B 0,C 180,E1 -2252.812,E2 -2252.812} C_VEL
LIN {X 0,Y 573.015,Z 324.887,A -85,B 0,C 180,E1 -2253.868,E2 -2253.868} C_VEL
LIN {X 0,Y 572.962,Z 320.939,A -85,B 0,C 180,E1 -2254.926,E2 -2254.926} C_VEL
LIN {X 0,Y 573.074,Z 315.844,A -85,B 0,C 180,E1 -2255.983,E2 -2255.983} C_VEL
LIN {X 0,Y 573.083,Z 309.461,A -85,B 0,C 180,E1 -2257.044,E2 -2257.044} C_VEL
LIN {X 0,Y 573.177,Z 301.487,A -85,B 0,C 180,E1 -2258.106,E2 -2258.106} C_VEL
LIN {X 0,Y 573.279,Z 293.346,A -85,B 0,C 180,E1 -2258.992,E2 -2258.992} C_VEL
LIN {X 0,Y 573.337,Z 283.37,A -85,B 0,C 180,E1 -2259.881,E2 -2259.881} C_VEL
LIN {X 0,Y 573.453,Z 273.554,A -85,B 0,C 180,E1 -2260.593,E2 -2260.593} C_VEL
LIN {X 0,Y 573.555,Z 262.756,A -85,B 0,C 180,E1 -2261.226,E2 -2261.226} C_VEL
LIN {X 0,Y 573.675,Z 250.145,A -85,B 0,C 180,E1 -2261.796,E2 -2261.796} C_VEL
LIN {X 0,Y 573.818,Z 237.886,A -85,B 0,C 180,E1 -2262.197,E2 -2262.197} C_VEL
LIN {X 0,Y 573.649,Z 229.55,A -85,B 0,C 180,E1 -2262.397,E2 -2262.397} C_VEL
LIN {X 0,Y 572.984,Z 225.524,A -85,B 0,C 180,E1 -2262.485,E2 -2262.485} C_VEL
LIN {X 0,Y 573.031,Z 219.461,A -85,B 0,C 180,E1 -2264.925,E2 -2264.925} C_VEL
LIN {X 0,Y 573.058,Z 212.275,A -85,B 0,C 180,E1 -2267.854,E2 -2267.854} C_VEL
LIN {X 0,Y 573.119,Z 205.089,A -85,B 0,C 180,E1 -2270.831,E2 -2270.831} C_VEL
LIN {X 0,Y 573.121,Z 197.902,A -85,B 0,C 180,E1 -2273.87,E2 -2273.87} C_VEL
LIN {X 0,Y 573.174,Z 191.859,A -85,B 0,C 180,E1 -2276.479,E2 -2276.479} C_VEL
LIN {X 0,Y 573.231,Z 185.065,A -85,B 0,C 180,E1 -2279.485,E2 -2279.485} C_VEL
LIN {X 0,Y 573.277,Z 179.029,A -85,B 0,C 180,E1 -2282.232,E2 -2282.232} C_VEL
LIN {X 0,Y 573.34,Z 173.573,A -85,B 0,C 180,E1 -2284.786,E2 -2284.786} C_VEL
LIN {X 0,Y 573.383,Z 168.709,A -85,B 0,C 180,E1 -2287.182,E2 -2287.182} C_VEL
LIN {X 0,Y 573.506,Z 164.304,A -85,B 0,C 180,E1 -2289.585,E2 -2289.585} C_VEL
LIN {X 0,Y 573.522,Z 160.767,A -85,B 0,C 180,E1 -2291.625,E2 -2291.625} C_VEL
LIN {X 0,Y 573.324,Z 159.12,A -85,B 0,C 180,E1 -2292.65,E2 -2292.65} C_VEL
LIN {X 0,Y 573.209,Z 158.584,A -85,B 0,C 180,E1 -2293.665,E2 -2293.665} C_VEL
LIN {X 0,Y 573.229,Z 158.582,A -85,B 0,C 180,E1 -2296.64,E2 -2296.64} C_VEL
LIN {X 0,Y 573.242,Z 158.577,A -85,B 0,C 180,E1 -2299.474,E2 -2299.474} C_VEL
LIN {X 0,Y 573.23,Z 158.578,A -85,B 0,C 180,E1 -2302.192,E2 -2302.192} C_VEL
LIN {X 0,Y 573.23,Z 158.578,A -85,B 0,C 180,E1 -2305.228,E2 -2305.228} C_VEL
LIN {X 0,Y 573.245,Z 158.574,A -85,B 0,C 180,E1 -2307.772,E2 -2307.772} C_VEL
LIN {X 0,Y 573.257,Z 158.581,A -85,B 0,C 180,E1 -2310.633,E2 -2310.633} C_VEL
LIN {X 0,Y 573.215,Z 158.58,A -85,B 0,C 180,E1 -2313.022,E2 -2313.022} C_VEL
LIN {X 0,Y 573.271,Z 158.57,A -85,B 0,C 180,E1 -2315.366,E2 -2315.366} C_VEL
LIN {X 0,Y 573.224,Z 158.585,A -85,B 0,C 180,E1 -2318.419,E2 -2318.419} C_VEL
LIN {X 0,Y 573.264,Z 158.574,A -85,B 0,C 180,E1 -2320.73,E2 -2320.73} C_VEL
LIN {X 0,Y 573.247,Z 158.575,A -85,B 0,C 180,E1 -2323.621,E2 -2323.621} C_VEL
LIN {X 0,Y 573.267,Z 158.576,A -85,B 0,C 180,E1 -2325.807,E2 -2325.807} C_VEL
LIN {X 0,Y 573.257,Z 158.573,A -85,B 0,C 180,E1 -2328.744,E2 -2328.744} C_VEL
LIN {X 0,Y 573.284,Z 158.572,A -85,B 0,C 180,E1 -2331.54,E2 -2331.54} C_VEL
LIN {X 0,Y 573.279,Z 158.572,A -85,B 0,C 180,E1 -2334.371,E2 -2334.371} C_VEL
LIN {X 0,Y 573.299,Z 158.574,A -85,B 0,C 180,E1 -2337.892,E2 -2337.892} C_VEL
LIN {X 0,Y 573.324,Z 158.564,A -85,B 0,C 180,E1 -2340.702,E2 -2340.702} C_VEL
LIN {X 0,Y 573.233,Z 158.584,A -85,B 0,C 180,E1 -2343.514,E2 -2343.514} C_VEL
LIN {X 0,Y 573.285,Z 158.577,A -85,B 0,C 180,E1 -2345.628,E2 -2345.628} C_VEL
LIN {X 0,Y 573.282,Z 158.569,A -85,B 0,C 180,E1 -2348.459,E2 -2348.459} C_VEL
LIN {X 0,Y 573.264,Z 158.581,A -85,B 0,C 180,E1 -2351.312,E2 -2351.312} C_VEL
LIN {X 0,Y 573.266,Z 158.571,A -85,B 0,C 180,E1 -2354.193,E2 -2354.193} C_VEL
LIN {X 0,Y 573.252,Z 158.582,A -85,B 0,C 180,E1 -2357.111,E2 -2357.111} C_VEL
LIN {X 0,Y 573.249,Z 158.573,A -85,B 0,C 180,E1 -2360.076,E2 -2360.076} C_VEL
LIN {X 0,Y 573.23,Z 158.576,A -85,B 0,C 180,E1 -2362.338,E2 -2362.338} C_VEL
LIN {X 0,Y 573.243,Z 158.576,A -85,B 0,C 180,E1 -2364.387,E2 -2364.387} C_VEL
LIN {X 0,Y 572.616,Z 158.662,A -85,B 0,C 180,E1 -2364.974,E2 -2364.974} C_VEL
LIN {X 0,Y 569.774,Z 159.015,A -85,B 0,C 180,E1 -2365.925,E2 -2365.925} C_VEL
LIN {X 0,Y 567.344,Z 159.316,A -85,B 0,C 180,E1 -2366.691,E2 -2366.691} C_VEL
LIN {X 0,Y 566.293,Z 159.444,A -85,B 0,C 180,E1 -2367.282,E2 -2367.282} C_VEL
LIN {X 0,Y 566.205,Z 159.452,A -85,B 0,C 180,E1 -2367.482,E2 -2367.482} C_VEL
LIN {X 0,Y 566.219,Z 159.449,A -85,B 0,C 180,E1 -2369.767,E2 -2369.767} C_VEL
LIN {X 0,Y 566.199,Z 159.456,A -85,B 0,C 180,E1 -2372.43,E2 -2372.43} C_VEL
LIN {X 0,Y 566.207,Z 159.455,A -85,B 0,C 180,E1 -2374.994,E2 -2374.994} C_VEL
LIN {X 0,Y 566.19,Z 159.453,A -85,B 0,C 180,E1 -2377.461,E2 -2377.461} C_VEL
LIN {X 0,Y 566.221,Z 159.454,A -85,B 0,C 180,E1 -2380.197,E2 -2380.197} C_VEL
LIN {X 0,Y 566.199,Z 159.453,A -85,B 0,C 180,E1 -2383.054,E2 -2383.054} C_VEL
LIN {X 0,Y 566.192,Z 159.458,A -85,B 0,C 180,E1 -2386.049,E2 -2386.049} C_VEL
LIN {X 0,Y 566.205,Z 159.452,A -85,B 0,C 180,E1 -2388.864,E2 -2388.864} C_VEL
LIN {X 0,Y 566.184,Z 159.456,A -85,B 0,C 180,E1 -2391.637,E2 -2391.637} C_VEL
LIN {X 0,Y 566.208,Z 159.456,A -85,B 0,C 180,E1 -2394.312,E2 -2394.312} C_VEL
LIN {X 0,Y 566.224,Z 159.448,A -85,B 0,C 180,E1 -2396.899,E2 -2396.899} C_VEL
LIN {X 0,Y 566.189,Z 159.455,A -85,B 0,C 180,E1 -2399.408,E2 -2399.408} C_VEL
LIN {X 0,Y 566.224,Z 159.458,A -85,B 0,C 180,E1 -2401.859,E2 -2401.859} C_VEL
LIN {X 0,Y 566.209,Z 159.453,A -85,B 0,C 180,E1 -2404.251,E2 -2404.251} C_VEL
LIN {X 0,Y 566.187,Z 159.453,A -85,B 0,C 180,E1 -2406.714,E2 -2406.714} C_VEL
LIN {X 0,Y 566.211,Z 159.459,A -85,B 0,C 180,E1 -2409.663,E2 -2409.663} C_VEL
LIN {X 0,Y 566.197,Z 159.453,A -85,B 0,C 180,E1 -2412.669,E2 -2412.669} C_VEL
LIN {X 0,Y 566.23,Z 159.455,A -85,B 0,C 180,E1 -2415.627,E2 -2415.627} C_VEL
LIN {X 0,Y 566.231,Z 159.449,A -85,B 0,C 180,E1 -2418.675,E2 -2418.675} C_VEL
LIN {X 0,Y 566.231,Z 159.455,A -85,B 0,C 180,E1 -2421.434,E2 -2421.434} C_VEL
LIN {X 0,Y 566.265,Z 159.444,A -85,B 0,C 180,E1 -2424.302,E2 -2424.302} C_VEL
LIN {X 0,Y 566.283,Z 159.442,A -85,B 0,C 180,E1 -2427.866,E2 -2427.866} C_VEL
LIN {X 0,Y 566.3,Z 159.445,A -85,B 0,C 180,E1 -2430.711,E2 -2430.711} C_VEL
LIN {X 0,Y 566.27,Z 159.452,A -85,B 0,C 180,E1 -2432.846,E2 -2432.846} C_VEL
LIN {X 0,Y 566.265,Z 159.444,A -85,B 0,C 180,E1 -2435.698,E2 -2435.698} C_VEL
LIN {X 0,Y 566.231,Z 159.455,A -85,B 0,C 180,E1 -2438.566,E2 -2438.566} C_VEL
LIN {X 0,Y 566.239,Z 159.448,A -85,B 0,C 180,E1 -2441.454,E2 -2441.454} C_VEL
LIN {X 0,Y 566.231,Z 159.457,A -85,B 0,C 180,E1 -2444.507,E2 -2444.507} C_VEL
LIN {X 0,Y 566.197,Z 159.453,A -85,B 0,C 180,E1 -2447.331,E2 -2447.331} C_VEL
LIN {X 0,Y 566.211,Z 159.459,A -85,B 0,C 180,E1 -2450.337,E2 -2450.337} C_VEL
LIN {X 0,Y 566.185,Z 159.453,A -85,B 0,C 180,E1 -2453.404,E2 -2453.404} C_VEL
LIN {X 0,Y 566.209,Z 159.453,A -85,B 0,C 180,E1 -2455.749,E2 -2455.749} C_VEL
LIN {X 0,Y 566.202,Z 159.46,A -85,B 0,C 180,E1 -2458.203,E2 -2458.203} C_VEL
LIN {X 0,Y 566.189,Z 159.455,A -85,B 0,C 180,E1 -2460.592,E2 -2460.592} C_VEL
LIN {X 0,Y 566.224,Z 159.448,A -85,B 0,C 180,E1 -2463.101,E2 -2463.101} C_VEL
LIN {X 0,Y 566.208,Z 159.456,A -85,B 0,C 180,E1 -2465.688,E2 -2465.688} C_VEL
LIN {X 0,Y 566.211,Z 159.451,A -85,B 0,C 180,E1 -2468.559,E2 -2468.559} C_VEL
LIN {X 0,Y 566.206,Z 159.452,A -85,B 0,C 180,E1 -2471.136,E2 -2471.136} C_VEL
LIN {X 0,Y 566.19,Z 159.457,A -85,B 0,C 180,E1 -2474.036,E2 -2474.036} C_VEL
LIN {X 0,Y 566.198,Z 159.454,A -85,B 0,C 180,E1 -2477.082,E2 -2477.082} C_VEL
LIN {X 0,Y 566.22,Z 159.454,A -85,B 0,C 180,E1 -2479.803,E2 -2479.803} C_VEL
LIN {X 0,Y 566.192,Z 159.452,A -85,B 0,C 180,E1 -2482.599,E2 -2482.599} C_VEL
LIN {X 0,Y 566.214,Z 159.456,A -85,B 0,C 180,E1 -2485.183,E2 -2485.183} C_VEL
LIN {X 0,Y 566.226,Z 159.451,A -85,B 0,C 180,E1 -2487.744,E2 -2487.744} C_VEL
LIN {X 0,Y 566.221,Z 159.449,A -85,B 0,C 180,E1 -2490.323,E2 -2490.323} C_VEL
LIN {X 0,Y 566.212,Z 159.453,A -85,B 0,C 180,E1 -2492.661,E2 -2492.661} C_VEL
LIN {X 0,Y 566.229,Z 159.457,A -85,B 0,C 180,E1 -2495.039,E2 -2495.039} C_VEL
LIN {X 0,Y 566.188,Z 159.453,A -85,B 0,C 180,E1 -2498.138,E2 -2498.138} C_VEL
LIN {X 0,Y 566.23,Z 159.453,A -85,B 0,C 180,E1 -2500.612,E2 -2500.612} C_VEL
LIN {X 0,Y 566.213,Z 159.451,A -85,B 0,C 180,E1 -2503.413,E2 -2503.413} C_VEL
LIN {X 0,Y 566.194,Z 159.456,A -85,B 0,C 180,E1 -2506.359,E2 -2506.359} C_VEL
LIN {X 0,Y 566.227,Z 159.457,A -85,B 0,C 180,E1 -2508.675,E2 -2508.675} C_VEL
LIN {X 0,Y 566.226,Z 159.448,A -85,B 0,C 180,E1 -2511.435,E2 -2511.435} C_VEL
LIN {X 0,Y 566.252,Z 159.451,A -85,B 0,C 180,E1 -2514.302,E2 -2514.302} C_VEL
LIN {X 0,Y 566.269,Z 159.445,A -85,B 0,C 180,E1 -2517.867,E2 -2517.867} C_VEL
LIN {X 0,Y 566.301,Z 159.442,A -85,B 0,C 180,E1 -2520.711,E2 -2520.711} C_VEL
LIN {X 0,Y 566.269,Z 159.444,A -85,B 0,C 180,E1 -2522.846,E2 -2522.846} C_VEL
LIN {X 0,Y 566.248,Z 159.448,A -85,B 0,C 180,E1 -2525.699,E2 -2525.699} C_VEL
LIN {X 0,Y 566.228,Z 159.45,A -85,B 0,C 180,E1 -2528.566,E2 -2528.566} C_VEL
LIN {X 0,Y 566.236,Z 159.449,A -85,B 0,C 180,E1 -2531.455,E2 -2531.455} C_VEL
LIN {X 0,Y 566.229,Z 159.449,A -85,B 0,C 180,E1 -2534.507,E2 -2534.507} C_VEL
LIN {X 0,Y 566.194,Z 159.455,A -85,B 0,C 180,E1 -2537.332,E2 -2537.332} C_VEL
LIN {X 0,Y 566.207,Z 159.452,A -85,B 0,C 180,E1 -2540.338,E2 -2540.338} C_VEL
LIN {X 0,Y 566.184,Z 159.459,A -85,B 0,C 180,E1 -2543.404,E2 -2543.404} C_VEL
LIN {X 0,Y 566.205,Z 159.457,A -85,B 0,C 180,E1 -2545.75,E2 -2545.75} C_VEL
LIN {X 0,Y 566.198,Z 159.452,A -85,B 0,C 180,E1 -2548.203,E2 -2548.203} C_VEL
LIN {X 0,Y 566.189,Z 159.457,A -85,B 0,C 180,E1 -2551.077,E2 -2551.077} C_VEL
LIN {X 0,Y 566.208,Z 159.454,A -85,B 0,C 180,E1 -2553.735,E2 -2553.735} C_VEL
LIN {X 0,Y 566.195,Z 159.454,A -85,B 0,C 180,E1 -2556.571,E2 -2556.571} C_VEL
LIN {X 0,Y 566.218,Z 159.453,A -85,B 0,C 180,E1 -2559.687,E2 -2559.687} C_VEL
LIN {X 0,Y 566.195,Z 159.461,A -85,B 0,C 180,E1 -2562.917,E2 -2562.917} C_VEL
LIN {X 0,Y 566.16,Z 159.463,A -85,B 0,C 180,E1 -2565.961,E2 -2565.961} C_VEL
LIN {X 0,Y 566.284,Z 160.019,A -85,B 0,C 180,E1 -2567.074,E2 -2567.074} C_VEL
LIN {X 0,Y 566.584,Z 163.381,A -85,B 0,C 180,E1 -2569.171,E2 -2569.171} C_VEL
LIN {X 0,Y 566.479,Z 167.82,A -85,B 0,C 180,E1 -2571.661,E2 -2571.661} C_VEL
LIN {X 0,Y 566.323,Z 172.762,A -85,B 0,C 180,E1 -2574.32,E2 -2574.32} C_VEL
LIN {X 0,Y 566.284,Z 178.141,A -85,B 0,C 180,E1 -2576.903,E2 -2576.903} C_VEL
LIN {X 0,Y 566.196,Z 183.53,A -85,B 0,C 180,E1 -2579.409,E2 -2579.409} C_VEL
LIN {X 0,Y 566.148,Z 188.92,A -85,B 0,C 180,E1 -2581.854,E2 -2581.854} C_VEL
LIN {X 0,Y 566.106,Z 194.309,A -85,B 0,C 180,E1 -2584.246,E2 -2584.246} C_VEL
LIN {X 0,Y 566.073,Z 200.05,A -85,B 0,C 180,E1 -2586.743,E2 -2586.743} C_VEL
LIN {X 0,Y 566.016,Z 206.885,A -85,B 0,C 180,E1 -2589.656,E2 -2589.656} C_VEL
LIN {X 0,Y 565.988,Z 212.275,A -85,B 0,C 180,E1 -2591.915,E2 -2591.915} C_VEL
LIN {X 0,Y 565.943,Z 219.461,A -85,B 0,C 180,E1 -2594.884,E2 -2594.884} C_VEL
LIN {X 0,Y 565.894,Z 225.524,A -85,B 0,C 180,E1 -2597.356,E2 -2597.356} C_VEL
LIN {X 0,Y 566.911,Z 232.502,A -85,B 0,C 180,E1 -2597.516,E2 -2597.516} C_VEL
LIN {X 0,Y 566.793,Z 245.127,A -85,B 0,C 180,E1 -2597.877,E2 -2597.877} C_VEL
LIN {X 0,Y 566.645,Z 257.464,A -85,B 0,C 180,E1 -2598.373,E2 -2598.373} C_VEL
LIN {X 0,Y 566.507,Z 269.827,A -85,B 0,C 180,E1 -2599.035,E2 -2599.035} C_VEL
LIN {X 0,Y 566.418,Z 281.083,A -85,B 0,C 180,E1 -2599.816,E2 -2599.816} C_VEL
LIN {X 0,Y 566.282,Z 289.583,A -85,B 0,C 180,E1 -2600.535,E2 -2600.535} C_VEL
LIN {X 0,Y 566.18,Z 298.389,A -85,B 0,C 180,E1 -2601.434,E2 -2601.434} C_VEL
LIN {X 0,Y 566.056,Z 307.007,A -85,B 0,C 180,E1 -2602.509,E2 -2602.509} C_VEL
LIN {X 0,Y 565.965,Z 313.872,A -85,B 0,C 180,E1 -2603.583,E2 -2603.583} C_VEL
LIN {X 0,Y 565.936,Z 319.364,A -85,B 0,C 180,E1 -2604.656,E2 -2604.656} C_VEL
LIN {X 0,Y 565.959,Z 323.666,A -85,B 0,C 180,E1 -2605.727,E2 -2605.727} C_VEL
LIN {X 0,Y 565.927,Z 325.964,A -85,B 0,C 180,E1 -2606.44,E2 -2606.44} C_VEL
LIN {X 0,Y 565.878,Z 327.795,A -85,B 0,C 180,E1 -2607.153,E2 -2607.153} C_VEL
LIN {X 0,Y 565.846,Z 330.189,A -85,B 0,C 180,E1 -2608.577,E2 -2608.577} C_VEL
LIN {X 0,Y 565.841,Z 330.782,A -85,B 0,C 180,E1 -2609.288,E2 -2609.288} C_VEL
LIN {X 0,Y 565.841,Z 330.782,A -85,B 0,C 180,E1 -2610.712,E2 -2610.712} C_VEL
LIN {X 0,Y 565.846,Z 330.189,A -85,B 0,C 180,E1 -2611.423,E2 -2611.423} C_VEL
LIN {X 0,Y 565.878,Z 327.795,A -85,B 0,C 180,E1 -2612.847,E2 -2612.847} C_VEL
LIN {X 0,Y 565.926,Z 324.883,A -85,B 0,C 180,E1 -2613.916,E2 -2613.916} C_VEL
LIN {X 0,Y 565.877,Z 320.934,A -85,B 0,C 180,E1 -2614.987,E2 -2614.987} C_VEL
LIN {X 0,Y 565.99,Z 315.839,A -85,B 0,C 180,E1 -2616.059,E2 -2616.059} C_VEL
LIN {X 0,Y 566.032,Z 309.456,A -85,B 0,C 180,E1 -2617.132,E2 -2617.132} C_VEL
LIN {X 0,Y 566.134,Z 301.489,A -85,B 0,C 180,E1 -2618.208,E2 -2618.208} C_VEL
LIN {X 0,Y 566.238,Z 293.348,A -85,B 0,C 180,E1 -2619.105,E2 -2619.105} C_VEL
LIN {X 0,Y 566.336,Z 283.364,A -85,B 0,C 180,E1 -2620.005,E2 -2620.005} C_VEL
LIN {X 0,Y 566.453,Z 273.546,A -85,B 0,C 180,E1 -2620.725,E2 -2620.725} C_VEL
LIN {X 0,Y 566.564,Z 262.758,A -85,B 0,C 180,E1 -2621.366,E2 -2621.366} C_VEL
LIN {X 0,Y 566.727,Z 250.149,A -85,B 0,C 180,E1 -2621.943,E2 -2621.943} C_VEL
LIN {X 0,Y 566.894,Z 237.87,A -85,B 0,C 180,E1 -2622.348,E2 -2622.348} C_VEL
LIN {X 0,Y 566.72,Z 230.409,A -85,B 0,C 180,E1 -2622.534,E2 -2622.534} C_VEL
LIN {X 0,Y 565.894,Z 225.524,A -85,B 0,C 180,E1 -2622.644,E2 -2622.644} C_VEL
LIN {X 0,Y 565.943,Z 219.461,A -85,B 0,C 180,E1 -2625.116,E2 -2625.116} C_VEL
LIN {X 0,Y 565.985,Z 212.275,A -85,B 0,C 180,E1 -2628.085,E2 -2628.085} C_VEL
LIN {X 0,Y 566.055,Z 205.089,A -85,B 0,C 180,E1 -2631.103,E2 -2631.103} C_VEL
LIN {X 0,Y 566.077,Z 197.902,A -85,B 0,C 180,E1 -2634.186,E2 -2634.186} C_VEL
LIN {X 0,Y 566.128,Z 192.293,A -85,B 0,C 180,E1 -2636.642,E2 -2636.642} C_VEL
LIN {X 0,Y 566.197,Z 185.327,A -85,B 0,C 180,E1 -2639.769,E2 -2639.769} C_VEL
LIN {X 0,Y 566.254,Z 179.548,A -85,B 0,C 180,E1 -2642.437,E2 -2642.437} C_VEL
LIN {X 0,Y 566.314,Z 174.137,A -85,B 0,C 180,E1 -2645.008,E2 -2645.008} C_VEL
LIN {X 0,Y 566.402,Z 169.469,A -85,B 0,C 180,E1 -2647.444,E2 -2647.444} C_VEL
LIN {X 0,Y 566.517,Z 165.318,A -85,B 0,C 180,E1 -2649.722,E2 -2649.722} C_VEL
LIN {X 0,Y 566.5,Z 161.631,A -85,B 0,C 180,E1 -2651.895,E2 -2651.895} C_VEL
LIN {X 0,Y 566.234,Z 159.828,A -85,B 0,C 180,E1 -2653.05,E2 -2653.05} C_VEL
LIN {X 0,Y 566.165,Z 159.465,A -85,B 0,C 180,E1 -2654.963,E2 -2654.963} C_VEL
LIN {X 0,Y 566.184,Z 159.455,A -85,B 0,C 180,E1 -2657.91,E2 -2657.91} C_VEL
LIN {X 0,Y 566.217,Z 159.458,A -85,B 0,C 180,E1 -2660.726,E2 -2660.726} C_VEL
